(* IEC 61131-3 sources: manufacturing_io/scenes (part 2) *)

(* ---- mps-sorting.st ---- *)
VAR
	START_EDGE : BOOL;
	PB_START_LAST : BOOL;
	STOP_REQ : BOOL;
	SEL_LAST : BOOL := TRUE;
	SEL_CHANGED : BOOL;
	T_WD : TON;
	T_READ : TON;
	T_FEED : TON;
	STEP_LAST : UDINT;
	KIND : UINT;
	NEXT_FEED : UINT;
	CLEAR : BOOL;
	RUNNING : BOOL;
	MEM_BELT : BOOL;
	MEM_STOP : BOOL;
	MEM_W1 : BOOL;
	MEM_W2 : BOOL;
	IND_BELT_LAST : BOOL;
	IND_STOP_LAST : BOOL;
	IND_W1_LAST : BOOL;
	IND_W2_LAST : BOOL;
	IND_ACTIVE : BOOL;
	ESTOP : BOOL;
	READY : BOOL;
	MASTER_ON : BOOL;
	HOMED : BOOL;
	MASTER_EDGE : BOOL;
	PB_MASTER_LAST : BOOL;
	HOME_EDGE : BOOL;
	PB_HOME_LAST : BOOL;
END_VAR
// mps-sorting: Festo Didactic's MPS Sorting station 8046325 (manual 8046391, 11/2015). The
// sequence and the IO are the manual's: a 40 mm workpiece is laid on the belt, a fork light
// barrier sees it, the belt runs it up to a stop, and three sensors at the stop say what it is -
// a through-beam sees every workpiece, a retro-reflective one sees every one that is NOT matt
// black, and an inductive one sees the metal. So black = seen but not by the retro one, red =
// retro but not inductive, metallic = both. Red goes to the chute at the belt START (Weiche 1),
// metallic to the one in the MIDDLE (Weiche 2), black runs off the belt END.
// The same sequence runs without a PLC in mps-sorting.ctl.js - keep the two in step.
//
// ONE difference from the real machine, deliberate: Festo's Q3 is "Stopper einfahren" - the stop
// is out by default and the output retracts it. Here the stop pops UP out of the belt
// (STOP_HOLD, energised to hold), because in this simulator a stop a part passes UNDER holds it
// from a positive distance (CLAUDE.md). It is the same signal inverted.
//
// KIND: 0 = black, 1 = red, 2 = metallic.

START_EDGE := PB_START AND NOT PB_START_LAST;
PB_START_LAST := PB_START;
IF PB_CSTOP THEN
	STOP_REQ := TRUE;
END_IF;
SEL_CHANGED := SEL_AUTO <> SEL_LAST;
SEL_LAST := SEL_AUTO;

ESTOP := PB_ESTOP;
MASTER_EDGE := PB_MASTER AND NOT PB_MASTER_LAST;
PB_MASTER_LAST := PB_MASTER;
HOME_EDGE := PB_HOME AND NOT PB_HOME_LAST;
PB_HOME_LAST := PB_HOME;
IF ESTOP THEN
	MASTER_ON := FALSE;
	HOMED := FALSE;
ELSIF MASTER_EDGE THEN
	MASTER_ON := TRUE;
END_IF;
READY := MASTER_ON AND NOT ESTOP;

// Everything laid on the belt has reached a bin: the invariant a discharge step waits for. A
// count that "has moved" cannot say WHICH workpiece moved (CLAUDE.md).
CLEAR := (EM_BLACK_CNT + EM_RED_CNT + EM_METAL_CNT) = (RM_1_CNT + RM_2_CNT + RM_3_CNT);

CASE ST1_STEP OF
	0:	// Ausgangsstellung: belt off, stop out, both gates in
		BELT_FWD := FALSE;
		W1_EXT := FALSE;
		W2_EXT := FALSE;
		EM_BLACK := FALSE;
		EM_RED := FALSE;
		EM_METAL := FALSE;
		STOP_HOLD := TRUE;
		IF START_EDGE AND SEL_AUTO AND READY AND HOMED THEN
			STOP_REQ := FALSE;
			ST1_STEP := 10;
		END_IF;
	10:	// the operator lays the next workpiece on the belt, one colour at a time
		BELT_FWD := FALSE;
		STOP_HOLD := TRUE;
		EM_BLACK := NEXT_FEED = 0;
		EM_RED := NEXT_FEED = 1;
		EM_METAL := NEXT_FEED = 2;
		IF T_FEED.Q THEN
			NEXT_FEED := (NEXT_FEED + 1) MOD 3;
			ST1_STEP := 15;
		END_IF;
	15:	// Startvoraussetzung: Werkstück am Bandanfang
		EM_BLACK := FALSE;
		EM_RED := FALSE;
		EM_METAL := FALSE;
		BELT_FWD := FALSE;
		STOP_HOLD := TRUE;
		IF WP_AT_START AND NOT CHUTE_FULL THEN
			ST1_STEP := 20;
		END_IF;
	20:	// Bandmotor ein
		BELT_FWD := TRUE;
		STOP_HOLD := TRUE;
		IF WP_DETECTED THEN
			ST1_STEP := 30;
		END_IF;
	30:	// Farb-/Materialidentifikation, with the workpiece held against the stop
		BELT_FWD := TRUE;
		IF T_READ.Q THEN
			IF WP_METALLIC THEN
				KIND := 2;
				ST1_STEP := 50;
			ELSIF WP_NOT_BLACK THEN
				KIND := 1;
				ST1_STEP := 40;
			ELSE
				KIND := 0;
				ST1_STEP := 60;
			END_IF;
		END_IF;
	40:	// red: Weiche 1 ausfahren
		BELT_FWD := TRUE;
		W1_EXT := TRUE;
		IF W1_OUT THEN
			ST1_STEP := 41;
		END_IF;
	41:	// Sperre einfahren
		BELT_FWD := TRUE;
		STOP_HOLD := FALSE;
		IF AS_STOP_FREE THEN
			ST1_STEP := 42;
		END_IF;
	42:	// Werkstück ausgeschleust
		BELT_FWD := TRUE;
		IF CLEAR THEN
			ST1_STEP := 43;
		END_IF;
	43:	// Weiche 1 einfahren
		BELT_FWD := TRUE;
		W1_EXT := FALSE;
		IF AS_W1_IN THEN
			ST1_STEP := 70;
		END_IF;
	50:	// metallic: Weiche 2 ausfahren
		BELT_FWD := TRUE;
		W2_EXT := TRUE;
		IF W2_OUT THEN
			ST1_STEP := 51;
		END_IF;
	51:
		BELT_FWD := TRUE;
		STOP_HOLD := FALSE;
		IF AS_STOP_FREE THEN
			ST1_STEP := 52;
		END_IF;
	52:
		BELT_FWD := TRUE;
		IF CLEAR THEN
			ST1_STEP := 53;
		END_IF;
	53:
		BELT_FWD := TRUE;
		W2_EXT := FALSE;
		IF AS_W2_IN THEN
			ST1_STEP := 70;
		END_IF;
	60:	// black: let it go, it runs off the belt end onto the third chute
		BELT_FWD := TRUE;
		STOP_HOLD := FALSE;
		IF AS_STOP_FREE THEN
			ST1_STEP := 61;
		END_IF;
	61:
		BELT_FWD := TRUE;
		IF CLEAR THEN
			ST1_STEP := 70;
		END_IF;
	70:	// Bandmotor aus, Sperre ausfahren
		BELT_FWD := FALSE;
		STOP_HOLD := TRUE;
		IF AS_STOP_HOLD THEN
			CYCLE_CNT := CYCLE_CNT + 1;
			IF STOP_REQ THEN
				ST1_STEP := 0;
			ELSE
				ST1_STEP := 10;
			END_IF;
		END_IF;
	800:	// HOME is the station's Ausgangsstellung
		BELT_FWD := FALSE;
		W1_EXT := FALSE;
		W2_EXT := FALSE;
		EM_BLACK := FALSE;
		EM_RED := FALSE;
		EM_METAL := FALSE;
		STOP_HOLD := TRUE;
		IF AS_STOP_HOLD AND AS_W1_IN AND AS_W2_IN THEN
			HOMED := TRUE;
			ST1_STEP := 0;
		END_IF;
	900:	// stuck, or the selector was turned while running
		BELT_FWD := FALSE;
		W1_EXT := FALSE;
		W2_EXT := FALSE;
		EM_BLACK := FALSE;
		EM_RED := FALSE;
		EM_METAL := FALSE;
		IF START_EDGE AND SEL_AUTO THEN
			STOP_REQ := FALSE;
			ST1_STEP := 0;
		END_IF;
	910:	// the master circuit is open: the stop KEEPS the workpiece it is holding
		BELT_FWD := FALSE;
		W1_EXT := FALSE;
		W2_EXT := FALSE;
		EM_BLACK := FALSE;
		EM_RED := FALSE;
		EM_METAL := FALSE;
		IF READY THEN
			ST1_STEP := 0;
		END_IF;
END_CASE;

RUNNING := ST1_STEP <> 0 AND ST1_STEP <> 800 AND ST1_STEP <> 900 AND ST1_STEP <> 910;

// TONs after the CASE: their Q is read by the NEXT scan.
T_READ(In := ST1_STEP = 30, PT := T#400ms);
T_FEED(In := ST1_STEP = 10, PT := T#600ms);

// Watchdog: a running step that stops moving is a jam, not patience - a workpiece taken off the
// belt by hand leaves step 20 waiting for a stop it will never reach. The TON is called BEFORE
// STEP_LAST is updated, so a step change gives it one scan of In = FALSE and resets it.
T_WD(In := ST1_STEP <> 0 AND ST1_STEP <> 900 AND ST1_STEP <> 910 AND ST1_STEP = STEP_LAST, PT := T#20s);
STEP_LAST := ST1_STEP;
IF T_WD.Q OR (SEL_CHANGED AND RUNNING) THEN
	ST1_STEP := 900;
	BELT_FWD := FALSE;
	W1_EXT := FALSE;
	W2_EXT := FALSE;
	EM_BLACK := FALSE;
	EM_RED := FALSE;
	EM_METAL := FALSE;
END_IF;

IF ESTOP THEN
	IF ST1_STEP <> 910 THEN
		ST1_STEP := 910;
	END_IF;
	BELT_FWD := FALSE;
	W1_EXT := FALSE;
	W2_EXT := FALSE;
	EM_BLACK := FALSE;
	EM_RED := FALSE;
	EM_METAL := FALSE;
ELSIF HOME_EDGE AND READY AND ST1_STEP = 0 THEN
	ST1_STEP := 800;
END_IF;

AUTO_RUN := ST1_STEP <> 0 AND ST1_STEP <> 800 AND ST1_STEP <> 900 AND ST1_STEP <> 910;
IND_ACTIVE := NOT SEL_AUTO AND NOT AUTO_RUN AND READY AND ST1_STEP <> 800;
IF IND_ACTIVE THEN
	IF IND_BELT AND NOT IND_BELT_LAST THEN
		MEM_BELT := NOT MEM_BELT;
	END_IF;
	IF IND_STOP AND NOT IND_STOP_LAST THEN
		MEM_STOP := NOT MEM_STOP;
	END_IF;
	IF IND_W1 AND NOT IND_W1_LAST THEN
		MEM_W1 := NOT MEM_W1;
	END_IF;
	IF IND_W2 AND NOT IND_W2_LAST THEN
		MEM_W2 := NOT MEM_W2;
	END_IF;
	BELT_FWD := MEM_BELT;
	STOP_HOLD := MEM_STOP;
	W1_EXT := MEM_W1;
	W2_EXT := MEM_W2;
	EM_BLACK := IND_FEED_BLACK;
	EM_RED := IND_FEED_RED;
	EM_METAL := IND_FEED_METAL;
ELSE
	MEM_BELT := FALSE;
	MEM_STOP := FALSE;
	MEM_W1 := FALSE;
	MEM_W2 := FALSE;
END_IF;
IND_BELT_LAST := IND_BELT;
IND_STOP_LAST := IND_STOP;
IND_W1_LAST := IND_W1;
IND_W2_LAST := IND_W2;

OVR := OVR_SET;
PL_START := AUTO_RUN;
PL_MASTER := MASTER_ON;
PL_HOME := HOMED;

(* ---- pallet-line.st ---- *)
VAR
	START_EDGE : BOOL;
	PB_START_LAST : BOOL;
	STOP_REQ : BOOL;
	SEL_LAST : BOOL := TRUE;
	SEL_CHANGED : BOOL;
	T_DWELL : TON;
	T_SETTLE : TON;
	T_CONF : TON;
	T_WD : TON;
	EM_P_LAST : UDINT;
	EM_W_LAST : UDINT;
	STEP_LAST : UDINT;
	GONE : UDINT;
	FED : UDINT;
	MEM_CV : BOOL;
	MEM_STOP : BOOL;
	MEM_LIFT : BOOL;
	IND_CV_LAST : BOOL;
	IND_STOP_LAST : BOOL;
	IND_LIFT_LAST : BOOL;
	ESTOP : BOOL;
	READY : BOOL;
	MASTER_ON : BOOL;
	HOMED : BOOL;
	MASTER_EDGE : BOOL;
	PB_MASTER_LAST : BOOL;
	HOME_EDGE : BOOL;
	PB_HOME_LAST : BOOL;
END_VAR
// pallet-line: a pallet is fed onto the belt, stopped at the station by a POP-UP stop, lifted off
// the belt and located square on its pins, loaded with a part, then put back down and released to
// the unloader. Repeat until CYCLE STOP. The same sequence runs without a PLC in pallet-line.ctl.js.
//
// The stop pops UP from under the belt on purpose. An overhead pin that the pallet has to drive
// under holds it from 7.9-15.1 mm away even after it has lifted clear and come to rest, and the
// clearance sweep is non-monotonic (5.1 held, 8.1 free, 11.1 free, 14.1 HELD, 17.1+ free), so
// there is no clearance to design to. Retracted, a pop-up stop is below the belt surface and
// nothing stands in the path at all.
//
// The pin must also be UP before a pallet arrives: one that rises under a pallet already over it
// tips the pallet off the belt (measured).
//
// The unloader counts the pallet AND the part riding on it, so the discharge step waits on both
// feeders: RM_CNT + GONE >= EM_P_CNT + EM_W_CNT.
//
// The panel has a selector AUTO / INDIVIDUAL (rb4axis): START only in AUTO, the individual buttons
// only in INDIVIDUAL, and a change while the sequence runs is a FAULT, not a pause.

START_EDGE := PB_START AND NOT PB_START_LAST;
PB_START_LAST := PB_START;
IF PB_CSTOP THEN
	STOP_REQ := TRUE;
END_IF;
SEL_CHANGED := SEL_AUTO <> SEL_LAST;
SEL_LAST := SEL_AUTO;

// The master circuit, as on the cell panel: E-STOP is a latching mushroom, MASTER ON energises
// the machine, and nothing runs without it. An E-STOP also loses the home position.
ESTOP := PB_ESTOP;
MASTER_EDGE := PB_MASTER AND NOT PB_MASTER_LAST;
PB_MASTER_LAST := PB_MASTER;
HOME_EDGE := PB_HOME AND NOT PB_HOME_LAST;
PB_HOME_LAST := PB_HOME;
IF ESTOP THEN
	MASTER_ON := FALSE;
	HOMED := FALSE;
ELSIF MASTER_EDGE THEN
	MASTER_ON := TRUE;
END_IF;
READY := MASTER_ON AND NOT ESTOP;

FED := EM_P_CNT + EM_W_CNT;
// A write-off goes STALE when what was written off turns up after all. GONE is a UDINT, so
// FED - RM_CNT with RM ahead underflows to about 4 billion: guard before you subtract.
IF RM_CNT >= FED THEN
	GONE := 0;
ELSIF RM_CNT + GONE > FED THEN
	GONE := FED - RM_CNT;
END_IF;

CASE ST1_STEP OF
	0:	// idle
		CV1_RUN := FALSE;
		EM_P_EMIT := FALSE;
		EM_W_EMIT := FALSE;
		SOL_LIFT := FALSE;
		SOL_STOP := FALSE;
		IF START_EDGE AND SEL_AUTO AND READY AND HOMED AND AS_LIFT_DN THEN
			STOP_REQ := FALSE;
			ST1_STEP := 10;
		END_IF;
	10:	// stop UP first, before any pallet is on its way
		SOL_STOP := TRUE;
		IF AS_STOP_UP THEN
			EM_P_LAST := EM_P_CNT;
			ST1_STEP := 20;
		END_IF;
	20:	// feed one pallet
		CV1_RUN := TRUE;
		EM_P_EMIT := TRUE;
		IF EM_P_CNT <> EM_P_LAST THEN
			EM_P_EMIT := FALSE;
			ST1_STEP := 30;
		END_IF;
	30:	// convey it to the station. The beam only says a pallet is HERE; the PIN locates it.
		// Stopping the belt on the beam edge left the pallet 106 mm short of the pin, so the
		// part feeder dropped its load onto the belt behind the deck every cycle (measured).
		CV1_RUN := TRUE;
		IF PE_STN THEN
			ST1_STEP := 35;
		END_IF;
	35:	// keep driving until it is pressed against the pin
		CV1_RUN := TRUE;
		IF T_SETTLE.Q THEN
			CV1_RUN := FALSE;
			ST1_STEP := 40;
		END_IF;
	40:	// lift and locate. The pallet must stay reported present for a CONFIRM time, not just for
		// the instant the switch first makes: a part is dropped on the strength of this signal,
		// and T_CONF restarts if it flickers.
		SOL_LIFT := TRUE;
		IF T_CONF.Q THEN
			EM_W_LAST := EM_W_CNT;
			ST1_STEP := 50;
		END_IF;
	50:	// load one part onto the pallet
		EM_W_EMIT := TRUE;
		IF EM_W_CNT <> EM_W_LAST THEN
			EM_W_EMIT := FALSE;
			ST1_STEP := 60;
		END_IF;
	60:	// the station does its work
		IF T_DWELL.Q THEN
			ST1_STEP := 70;
		END_IF;
	70:	// pallet back onto the belt
		SOL_LIFT := FALSE;
		IF AS_LIFT_DN THEN
			ST1_STEP := 80;
		END_IF;
	80:	// only now is the pin allowed down, clear of the path
		SOL_STOP := FALSE;
		IF AS_STOP_DN THEN
			ST1_STEP := 90;
		END_IF;
	90:	// discharge: every pallet and part fed must have reached the unloader
		CV1_RUN := TRUE;
		IF RM_CNT + GONE >= FED THEN
			CV1_RUN := FALSE;
			ST1_STEP := 100;
		END_IF;
	100:	// cycle complete
		CYCLE_CNT := CYCLE_CNT + 1;
		IF STOP_REQ THEN
			ST1_STEP := 0;
		ELSE
			ST1_STEP := 10;
		END_IF;
	800:	// HOME: the lift down and the pin down, so the belt is clear along its whole length
		CV1_RUN := FALSE;
		EM_P_EMIT := FALSE;
		EM_W_EMIT := FALSE;
		SOL_LIFT := FALSE;
		SOL_STOP := FALSE;
		IF AS_LIFT_DN AND AS_STOP_DN THEN
			HOMED := TRUE;
			ST1_STEP := 0;
		END_IF;
	910:	// E-STOP: the master circuit is open, so every solenoid de-energises - a 5/2 single-
		// solenoid valve springs back. The LIFT is the exception: it is a holder, and a real
		// machine does not drop what it carries when the power goes.
		CV1_RUN := FALSE;
		EM_P_EMIT := FALSE;
		EM_W_EMIT := FALSE;
		SOL_STOP := FALSE;
		IF READY THEN	// MASTER ON after the mushroom is released
			ST1_STEP := 0;
		END_IF;
	900:	// FAULT: a step stopped moving. Stop feeding and the belt; the pin keeps holding the
		// queue back and the lift keeps its pallet.
		CV1_RUN := FALSE;
		EM_P_EMIT := FALSE;
		EM_W_EMIT := FALSE;
		IF START_EDGE AND SEL_AUTO THEN
			STOP_REQ := FALSE;
			// Acknowledging writes off what never reached the unloader. Only HERE: at every START
			// it would write off pallets still legitimately on the belt.
			GONE := FED - RM_CNT;
			ST1_STEP := 0;
		END_IF;
END_CASE;

T_DWELL(In := (ST1_STEP = 60), PT := T#500ms);
// 106 mm from the beam edge to the pin at 250 mm/s is 424 ms; 700 leaves margin to press up.
T_SETTLE(In := (ST1_STEP = 35), PT := T#700ms);
T_CONF(In := (ST1_STEP = 40) AND AS_LIFT_UP AND PLT_PRESENT, PT := T#300ms);

// Watchdog: a running step that stops moving is a jam, not patience. Without it the sequence waits
// for ever and the machine only LOOKS alive. A selector change while running trips the same way.
T_WD(In := (ST1_STEP = STEP_LAST) AND (ST1_STEP <> 0) AND (ST1_STEP <> 900) AND (ST1_STEP <> 910), PT := T#15s);
IF ST1_STEP <> STEP_LAST THEN
	STEP_LAST := ST1_STEP;
END_IF;
IF T_WD.Q OR (SEL_CHANGED AND (ST1_STEP <> 0) AND (ST1_STEP <> 900) AND (ST1_STEP <> 910)) THEN
	ST1_STEP := 900;
	CV1_RUN := FALSE;
	EM_P_EMIT := FALSE;
	EM_W_EMIT := FALSE;
END_IF;

// E-STOP at any moment, and the HOME button when the machine is energised and idle.
IF ESTOP THEN
	IF ST1_STEP <> 910 THEN
		ST1_STEP := 910;
	END_IF;
	CV1_RUN := FALSE;
	EM_P_EMIT := FALSE;
	EM_W_EMIT := FALSE;
	SOL_STOP := FALSE;
ELSIF HOME_EDGE AND READY AND (ST1_STEP = 0) THEN
	ST1_STEP := 800;
END_IF;

AUTO_RUN := (ST1_STEP <> 0) AND (ST1_STEP <> 800) AND (ST1_STEP <> 900) AND (ST1_STEP <> 910);

// Individual operation: the buttons are momentary; the PLC keeps a toggle memory per actuator and
// clears it when INDIVIDUAL ends, so nothing stays latched into AUTO.
IF NOT SEL_AUTO AND NOT AUTO_RUN AND READY AND (ST1_STEP <> 800) THEN
	IF IND_CV AND NOT IND_CV_LAST THEN
		MEM_CV := NOT MEM_CV;
	END_IF;
	IF IND_STOP AND NOT IND_STOP_LAST THEN
		MEM_STOP := NOT MEM_STOP;
	END_IF;
	IF IND_LIFT AND NOT IND_LIFT_LAST THEN
		MEM_LIFT := NOT MEM_LIFT;
	END_IF;
	CV1_RUN := MEM_CV;
	SOL_STOP := MEM_STOP;
	SOL_LIFT := MEM_LIFT;
	EM_P_EMIT := IND_FEED_P;
	EM_W_EMIT := IND_FEED_W;
ELSE
	MEM_CV := FALSE;
	MEM_STOP := FALSE;
	MEM_LIFT := FALSE;
END_IF;
IND_CV_LAST := IND_CV;
IND_STOP_LAST := IND_STOP;
IND_LIFT_LAST := IND_LIFT;

// The speed override the operator dialled in, passed on to the axes and the belts.
OVR := OVR_SET;

PL_START := AUTO_RUN;
PL_MASTER := MASTER_ON;
PL_HOME := HOMED;

(* ---- palletizing.st ---- *)
VAR
	START_EDGE : BOOL;
	PB_START_LAST : BOOL;
	STOP_REQ : BOOL;
	SEL_LAST : BOOL := TRUE;
	SEL_CHANGED : BOOL;
	ESTOP : BOOL;
	READY : BOOL;
	MASTER_ON : BOOL;
	HOMED : BOOL;
	MASTER_EDGE : BOOL;
	PB_MASTER_LAST : BOOL;
	HOME_EDGE : BOOL;
	PB_HOME_LAST : BOOL;
	RUNNING : BOOL;
	LOAD_BUSY : BOOL;
	UNLOAD_BUSY : BOOL;
	LOAD_IDX : INT;
	UNLOAD_IDX : INT;
	FULL : ARRAY[0..3] OF BOOL;
	HALF : BOOL;
	ROW_Y : LREAL := 330.0;
	PICKED : BOOL;
	ANY_VAC : BOOL;
	NO_VAC : BOOL;
	NO_UVAC : BOOL;
	NEED_FILL : BOOL := TRUE;
	PAL_BASE : UDINT;
	NEXT_ST : INT;
	T_FILL : TON;
	T_PICK : TON;
	T_UPICK : TON;
	T_WD1 : TON;
	T_WD2 : TON;
	T_WD3 : TON;
	STEP1_LAST : UDINT;
	STEP2_LAST : UDINT;
	STEP3_LAST : UDINT;
	JAM : BOOL;
	MEM_VAC : BOOL;
	IND_VAC_LAST : BOOL;
	MEM_LIFT : BOOL;
	IND_LIFT_LAST : BOOL;
	MEM_PAL : BOOL;
	IND_PAL_LAST : BOOL;
	MEM_JIG : BOOL;
	IND_JIG_LAST : BOOL;
	MEM_UVAC : BOOL;
	IND_UVAC_LAST : BOOL;
	MEM_ULIFT : BOOL;
	IND_ULIFT_LAST : BOOL;
	MEM_USHIFT : BOOL;
	IND_USHIFT_LAST : BOOL;
	INDIVIDUAL : BOOL;
END_VAR
// palletizing: a 10 x 10 pallet of spark plugs, a five-up vacuum gantry on two servo axes, a
// rotary carrier of five-slot jigs, and an unload head that hands the plugs to the next process.
// The same sequence runs without a PLC in palletizing.ctl.js.
//
// THREE stations run at the same time, which is what a cell does and what one long sequence could
// not: the gantry goes back for the next five as soon as it has put its five down, while the
// carrier indexes and the unloader empties a jig on the far side. They meet at the carrier: FULL[i]
// says which jig has parts in it, and neither head lets the table turn under it.
//
// A head takes what is there. A hole may be empty - a plug was lifted out, or the pallet is
// finished - and the gantry carries on with what it got rather than waiting for a plug that is not
// coming. Nothing at all means the tray is empty, and a fresh pallet is called for.
//
// Gantry positions are millimetres on each axis, measured from the scene: cup 3 sits at
// X = GX - 300 and Y = GY - 600, so the pallet halves are at GX 150 and 450, the jig at GX 1268,
// and pallet row r is at GY 330 + 60 r.

START_EDGE := PB_START AND NOT PB_START_LAST;
PB_START_LAST := PB_START;
IF PB_CSTOP THEN
	STOP_REQ := TRUE;
END_IF;
SEL_CHANGED := SEL_AUTO <> SEL_LAST;
SEL_LAST := SEL_AUTO;

// The master circuit: E-STOP is a latching mushroom, MASTER ON energises the machine, and an
// E-STOP also loses the home position.
ESTOP := PB_ESTOP;
MASTER_EDGE := PB_MASTER AND NOT PB_MASTER_LAST;
PB_MASTER_LAST := PB_MASTER;
HOME_EDGE := PB_HOME AND NOT PB_HOME_LAST;
PB_HOME_LAST := PB_HOME;
IF ESTOP THEN
	MASTER_ON := FALSE;
	HOMED := FALSE;
ELSIF MASTER_EDGE THEN
	MASTER_ON := TRUE;
END_IF;
READY := MASTER_ON AND NOT ESTOP;

ANY_VAC := VAC_SW1 OR VAC_SW2 OR VAC_SW3 OR VAC_SW4 OR VAC_SW5;
NO_VAC := NOT ANY_VAC;
NO_UVAC := NOT (UVAC_SW1 OR UVAC_SW2 OR UVAC_SW3 OR UVAC_SW4 OR UVAC_SW5);
// The jig standing at the load station, and the one at the unload station.
LOAD_IDX := (2 - TBL_STATION + 4) MOD 4;
UNLOAD_IDX := (4 - TBL_STATION) MOD 4;
// Neither head lets the carrier turn while it is over a jig.
LOAD_BUSY := (ST1_STEP >= 57) AND (ST1_STEP <= 80);
UNLOAD_BUSY := (ST3_STEP >= 110) AND (ST3_STEP <= 130);

// ---------------------------------------------------------------- ST1: the depalletiser
CASE ST1_STEP OF
	0:	// idle: head up, vacuum off
		VAC_ON := FALSE;
		GX_EXEC := FALSE;
		GY_EXEC := FALSE;
		SOL_Z_DN := FALSE;
		SOL_Z_UP := TRUE;
		EM_PAL_EN := FALSE;
		IF START_EDGE AND SEL_AUTO AND READY AND HOMED AND AS_Z_UP AND AS_U_UP THEN
			STOP_REQ := FALSE;
			ST2_STEP := 10;
			ST3_STEP := 100;
			IF NEED_FILL THEN
				PAL_BASE := EM_PAL_CNT;
				ST1_STEP := 5;
			ELSE
				ST1_STEP := 10;
			END_IF;
		END_IF;
	5:	// A fresh pallet. The tray is FULL when the loader stops delivering, not after a count of
		// 100: a hole that still had a plug in it would make a count wait for ever.
		PAL_CLAMP := TRUE;
		EM_PAL_EN := TRUE;
		IF EM_PAL_CNT <> PAL_BASE THEN
			PAL_BASE := EM_PAL_CNT;
		ELSIF T_FILL.Q THEN
			EM_PAL_EN := FALSE;
			NEED_FILL := FALSE;
			ST1_STEP := 10;
		END_IF;
	10:	// both gantry axes move at once; Execute is a LEVEL held until Done
		PAL_CLAMP := TRUE;
		JIG_CLAMP := TRUE;
		IF HALF THEN
			GX_TGT := 450.0;
		ELSE
			GX_TGT := 150.0;
		END_IF;
		GY_TGT := ROW_Y;
		GX_EXEC := TRUE;
		GY_EXEC := TRUE;
		IF GX_DONE AND GY_DONE THEN
			GX_EXEC := FALSE;
			GY_EXEC := FALSE;
			ST1_STEP := 15;
		END_IF;
	15:	// wait until the plant has seen Execute drop
		IF NOT GX_DONE AND NOT GY_DONE THEN
			ST1_STEP := 20;
		END_IF;
	20:	// head down onto the row
		SOL_Z_UP := FALSE;
		SOL_Z_DN := TRUE;
		IF AS_Z_DN THEN
			ST1_STEP := 30;
		END_IF;
	30:	// the tray lets go while the cups take whatever is there
		PAL_CLAMP := FALSE;
		VAC_ON := TRUE;
		IF T_PICK.Q THEN
			PICKED := ANY_VAC;
			ST1_STEP := 40;
		END_IF;
	40:	// the tray is held again, and the head lifts with what it got
		PAL_CLAMP := TRUE;
		SOL_Z_DN := FALSE;
		SOL_Z_UP := TRUE;
		IF AS_Z_UP THEN
			IF PICKED THEN
				ST1_STEP := 50;
			ELSE
				// nothing at all came up: the tray is empty
				NEED_FILL := TRUE;
				PAL_BASE := EM_PAL_CNT;
				ST1_STEP := 5;
			END_IF;
		END_IF;
	50:	// across to the jig at the load station
		GX_TGT := 1268.0;
		GY_TGT := 600.0;
		GX_EXEC := TRUE;
		GY_EXEC := TRUE;
		IF GX_DONE AND GY_DONE THEN
			GX_EXEC := FALSE;
			GY_EXEC := FALSE;
			ST1_STEP := 55;
		END_IF;
	55:	// wait until the plant has seen Execute drop
		IF NOT GX_DONE AND NOT GY_DONE THEN
			ST1_STEP := 57;
		END_IF;
	57:	// the load station must be standing still with an empty jig under it
		IF TBL_INPOS AND NOT FULL[LOAD_IDX] THEN
			ST1_STEP := 60;
		END_IF;
	60:	// head down over the jig
		SOL_Z_UP := FALSE;
		SOL_Z_DN := TRUE;
		IF AS_Z_DN THEN
			ST1_STEP := 70;
		END_IF;
	70:	// the jig nests take the plugs as the cups let go: one part, one holder
		VAC_ON := FALSE;
		IF NO_VAC THEN
			ST1_STEP := 80;
		END_IF;
	80:	// head up; the carrier may take this jig away now
		SOL_Z_DN := FALSE;
		SOL_Z_UP := TRUE;
		IF AS_Z_UP THEN
			FULL[LOAD_IDX] := TRUE;
			CYCLE_CNT := CYCLE_CNT + 1;
			IF HALF THEN
				HALF := FALSE;
				IF ROW_Y >= 870.0 THEN
					ROW_Y := 330.0;
					NEED_FILL := TRUE;
				ELSE
					ROW_Y := ROW_Y + 60.0;
				END_IF;
			ELSE
				HALF := TRUE;
			END_IF;
			IF STOP_REQ THEN
				ST1_STEP := 0;
			ELSIF NEED_FILL THEN
				PAL_BASE := EM_PAL_CNT;
				ST1_STEP := 5;
			ELSE
				ST1_STEP := 10;
			END_IF;
		END_IF;
	800:	// HOME: heads up, unload shift over the jig, both gantry axes to zero, carrier to its
		// origin. The vacuum is left alone: a head keeps the plugs it is holding.
		TBL_RUN := NOT TBL_ORIGIN;
		SOL_Z_DN := FALSE;
		SOL_Z_UP := TRUE;
		SOL_U_DN := FALSE;
		SOL_U_UP := TRUE;
		SOL_U_BIN := FALSE;
		SOL_U_JIG := TRUE;
		GX_TGT := 0.0;
		GY_TGT := 0.0;
		GX_EXEC := TRUE;
		GY_EXEC := TRUE;
		IF AS_Z_UP AND AS_U_UP AND AS_U_JIG AND GX_DONE AND GY_DONE AND TBL_ORIGIN THEN
			GX_EXEC := FALSE;
			GY_EXEC := FALSE;
			TBL_RUN := FALSE;
			HOMED := TRUE;
			ST1_STEP := 0;
		END_IF;
	900:	// FAULT: stuck, or the selector was turned while running. Motion and feeding off; the
		// trays and the cups keep whatever they hold.
		TBL_RUN := FALSE;
		GX_EXEC := FALSE;
		GY_EXEC := FALSE;
		EM_PAL_EN := FALSE;
		PAL_CLAMP := TRUE;
		JIG_CLAMP := TRUE;
		IF START_EDGE AND SEL_AUTO THEN
			STOP_REQ := FALSE;
			ST1_STEP := 0;
		END_IF;
	910:	// E-STOP: the master circuit is open, so every solenoid de-energises - which is what
		// really happens: a 5/2 single-solenoid valve springs back, a double one holds. The trays
		// and the cups KEEP their parts: a hundred plugs let loose in their pockets is not what a
		// power cut does, and it costs the plant four times the work.
		TBL_RUN := FALSE;
		GX_EXEC := FALSE;
		GY_EXEC := FALSE;
		EM_PAL_EN := FALSE;
		SOL_Z_DN := FALSE;
		SOL_Z_UP := FALSE;
		SOL_U_DN := FALSE;
		SOL_U_UP := FALSE;
		SOL_U_BIN := FALSE;
		SOL_U_JIG := FALSE;
		PAL_CLAMP := TRUE;
		JIG_CLAMP := TRUE;
		IF READY THEN	// MASTER ON after the mushroom is released
			ST1_STEP := 0;
		END_IF;
END_CASE;

RUNNING := (ST1_STEP <> 0) AND (ST1_STEP <> 800) AND (ST1_STEP <> 900) AND (ST1_STEP <> 910);

// ---------------------------------------------------------------- ST2: the jig carrier
IF NOT RUNNING THEN
	ST2_STEP := 0;
	TBL_RUN := FALSE;
ELSE
	CASE ST2_STEP OF
		10:	// Turn when there is a full jig to move on AND an empty one to bring to the unloader,
			// and never while a head is over the table.
			TBL_RUN := FALSE;
			IF FULL[LOAD_IDX] AND NOT FULL[UNLOAD_IDX] AND NOT LOAD_BUSY AND NOT UNLOAD_BUSY AND TBL_INPOS THEN
				NEXT_ST := (TBL_STATION + 1) MOD 4;
				ST2_STEP := 20;
			END_IF;
		20:	// the invariant: this index has landed on the station it was sent to
			TBL_RUN := TRUE;
			IF TBL_INPOS AND (TBL_STATION = NEXT_ST) THEN
				TBL_RUN := FALSE;
				ST2_STEP := 10;
			END_IF;
		ELSE
			ST2_STEP := 10;
	END_CASE;
END_IF;

// ---------------------------------------------------------------- ST3: the unloader
IF NOT RUNNING THEN
	ST3_STEP := 0;
ELSE
	CASE ST3_STEP OF
		100:	// wait for a full jig to arrive and stand still
			IF FULL[UNLOAD_IDX] AND TBL_INPOS THEN
				ST3_STEP := 110;
			END_IF;
		110:	// over the jig
			SOL_U_BIN := FALSE;
			SOL_U_JIG := TRUE;
			IF AS_U_JIG THEN
				ST3_STEP := 115;
			END_IF;
		115:	// down onto it
			SOL_U_UP := FALSE;
			SOL_U_DN := TRUE;
			IF AS_U_DN THEN
				ST3_STEP := 120;
			END_IF;
		120:	// whatever is in the jig, however many: a gap is not a reason to stop
			JIG_CLAMP := FALSE;
			UVAC_ON := TRUE;
			IF T_UPICK.Q THEN
				ST3_STEP := 130;
			END_IF;
		130:	// up, and the carrier is free to turn again
			JIG_CLAMP := TRUE;
			SOL_U_DN := FALSE;
			SOL_U_UP := TRUE;
			IF AS_U_UP THEN
				FULL[UNLOAD_IDX] := FALSE;
				ST3_STEP := 140;
			END_IF;
		140:	// across to the next process
			SOL_U_JIG := FALSE;
			SOL_U_BIN := TRUE;
			IF AS_U_BIN THEN
				ST3_STEP := 150;
			END_IF;
		150:	// down over the bin
			SOL_U_UP := FALSE;
			SOL_U_DN := TRUE;
			IF AS_U_DN THEN
				ST3_STEP := 160;
			END_IF;
		160:	// let them go: the next process takes them from here
			UVAC_ON := FALSE;
			IF NO_UVAC THEN
				ST3_STEP := 170;
			END_IF;
		170:	// up
			SOL_U_DN := FALSE;
			SOL_U_UP := TRUE;
			IF AS_U_UP THEN
				ST3_STEP := 180;
			END_IF;
		180:	// back over the jig, ready for the next one
			SOL_U_BIN := FALSE;
			SOL_U_JIG := TRUE;
			IF AS_U_JIG THEN
				ST3_STEP := 100;
			END_IF;
		ELSE
			ST3_STEP := 100;
	END_CASE;
END_IF;

// The loader drops one every 40 ms while it can, so 600 ms of nothing means the tray is full.
T_FILL(In := (ST1_STEP = 5) AND (EM_PAL_CNT = PAL_BASE), PT := T#600ms);
// A head is given this long to get hold of what is under it, then carries on with what it has.
T_PICK(In := (ST1_STEP = 30), PT := T#600ms);
T_UPICK(In := (ST3_STEP = 120), PT := T#600ms);

// Watchdog, one per station: a running step that stops moving is a jam, not patience. The
// carrier's wait for work and the unloader's wait for a jig are not stuck, so they are excluded.
T_WD1(In := (ST1_STEP = STEP1_LAST) AND RUNNING, PT := T#15s);
T_WD2(In := (ST2_STEP = STEP2_LAST) AND RUNNING AND (ST2_STEP <> 10), PT := T#15s);
T_WD3(In := (ST3_STEP = STEP3_LAST) AND RUNNING AND (ST3_STEP <> 100), PT := T#15s);
IF ST1_STEP <> STEP1_LAST THEN
	STEP1_LAST := ST1_STEP;
END_IF;
IF ST2_STEP <> STEP2_LAST THEN
	STEP2_LAST := ST2_STEP;
END_IF;
IF ST3_STEP <> STEP3_LAST THEN
	STEP3_LAST := ST3_STEP;
END_IF;
JAM := T_WD1.Q OR T_WD2.Q OR T_WD3.Q;
IF RUNNING AND (JAM OR SEL_CHANGED) THEN
	ST1_STEP := 900;
	ST2_STEP := 0;
	ST3_STEP := 0;
	TBL_RUN := FALSE;
	GX_EXEC := FALSE;
	GY_EXEC := FALSE;
	EM_PAL_EN := FALSE;
END_IF;

// E-STOP at any moment, and the HOME button when the machine is energised and idle.
IF ESTOP THEN
	IF ST1_STEP <> 910 THEN
		ST1_STEP := 910;
	END_IF;
	ST2_STEP := 0;
	ST3_STEP := 0;
	TBL_RUN := FALSE;
	GX_EXEC := FALSE;
	GY_EXEC := FALSE;
	EM_PAL_EN := FALSE;
	SOL_Z_DN := FALSE;
	SOL_Z_UP := FALSE;
	SOL_U_DN := FALSE;
	SOL_U_UP := FALSE;
	SOL_U_BIN := FALSE;
	SOL_U_JIG := FALSE;
	PAL_CLAMP := TRUE;
	JIG_CLAMP := TRUE;
ELSIF HOME_EDGE AND READY AND (ST1_STEP = 0) THEN
	ST1_STEP := 800;
END_IF;

AUTO_RUN := (ST1_STEP <> 0) AND (ST1_STEP <> 800) AND (ST1_STEP <> 900) AND (ST1_STEP <> 910);

// Individual operation: momentary buttons, a PLC toggle memory per actuator, cleared when
// INDIVIDUAL ends. The index button is held and the carrier turns while it is down.
INDIVIDUAL := NOT SEL_AUTO AND NOT AUTO_RUN AND READY AND (ST1_STEP <> 800);
IF INDIVIDUAL THEN
	IF IND_VAC AND NOT IND_VAC_LAST THEN
		MEM_VAC := NOT MEM_VAC;
	END_IF;
	IF IND_LIFT AND NOT IND_LIFT_LAST THEN
		MEM_LIFT := NOT MEM_LIFT;
	END_IF;
	IF IND_PAL AND NOT IND_PAL_LAST THEN
		MEM_PAL := NOT MEM_PAL;
	END_IF;
	IF IND_JIG AND NOT IND_JIG_LAST THEN
		MEM_JIG := NOT MEM_JIG;
	END_IF;
	IF IND_UVAC AND NOT IND_UVAC_LAST THEN
		MEM_UVAC := NOT MEM_UVAC;
	END_IF;
	IF IND_ULIFT AND NOT IND_ULIFT_LAST THEN
		MEM_ULIFT := NOT MEM_ULIFT;
	END_IF;
	IF IND_USHIFT AND NOT IND_USHIFT_LAST THEN
		MEM_USHIFT := NOT MEM_USHIFT;
	END_IF;
	VAC_ON := MEM_VAC;
	UVAC_ON := MEM_UVAC;
	PAL_CLAMP := MEM_PAL;
	JIG_CLAMP := MEM_JIG;
	SOL_Z_DN := MEM_LIFT;
	SOL_Z_UP := NOT MEM_LIFT;
	SOL_U_DN := MEM_ULIFT;
	SOL_U_UP := NOT MEM_ULIFT;
	SOL_U_BIN := MEM_USHIFT;
	SOL_U_JIG := NOT MEM_USHIFT;
	TBL_RUN := IND_INDEX;
ELSE
	MEM_VAC := FALSE;
	MEM_LIFT := FALSE;
	MEM_PAL := FALSE;
	MEM_JIG := FALSE;
	MEM_UVAC := FALSE;
	MEM_ULIFT := FALSE;
	MEM_USHIFT := FALSE;
END_IF;
IND_VAC_LAST := IND_VAC;
IND_LIFT_LAST := IND_LIFT;
IND_PAL_LAST := IND_PAL;
IND_JIG_LAST := IND_JIG;
IND_UVAC_LAST := IND_UVAC;
IND_ULIFT_LAST := IND_ULIFT;
IND_USHIFT_LAST := IND_USHIFT;

// The speed override the operator dialled in, passed on to the axes and the belts.
OVR := OVR_SET;

// Jog: the axis creeps while the button is held, and only on INDIVIDUAL.
GX_JOG_P := INDIVIDUAL AND IND_GX_P;
GX_JOG_N := INDIVIDUAL AND IND_GX_N;
GY_JOG_P := INDIVIDUAL AND IND_GY_P;
GY_JOG_N := INDIVIDUAL AND IND_GY_N;

PL_START := AUTO_RUN;
PL_MASTER := MASTER_ON;
PL_HOME := HOMED;

(* ---- pick-place.st ---- *)
VAR
	START_EDGE : BOOL;
	PB_START_LAST : BOOL;
	STOP_REQ : BOOL;
	T_WD : TON;
	EM_LAST : UDINT;
	STEP_LAST : UDINT;
	GONE : UDINT;
END_VAR
// pick-place: feed a part into the pick nest, pick it with the vacuum cup on the lift cylinder,
// traverse on the servo, lay it on the running outfeed belt, and come home while the belt takes
// it to the unloader. Repeat until STOP. The same sequence runs without a PLC in
// pick-place.ctl.js.
//
// Two handshakes matter. The servo's Execute is a LEVEL held until Done, and Done must be seen
// to drop before the next Execute. The nest clamp must open BEFORE the cup can take the part:
// one part is held by one holder.
//
// Waiting steps wait for an INVARIANT, not for a counter to move: a change cannot say which
// part moved (measured on a-to-b against the simulator: parts piled up, then pipelined).

START_EDGE := PB_START AND NOT PB_START_LAST;
PB_START_LAST := PB_START;
IF PB_STOP THEN
	STOP_REQ := TRUE;
END_IF;

// A write-off goes STALE when the part turns up after all, and then RM + GONE runs PAST EM and
// step 130 stops waiting at all. GONE is a UDINT, so EM_CNT - RM_CNT with RM ahead underflows to
// about 4 billion: guard before you subtract.
IF RM_CNT >= EM_CNT THEN
	GONE := 0;
ELSIF RM_CNT + GONE > EM_CNT THEN
	GONE := EM_CNT - RM_CNT;
END_IF;

CASE ST1_STEP OF
	0:	// idle
		CV_RUN := FALSE;
		EM_EMIT := FALSE;
		VAC_ON := FALSE;
		SOL_Z_DN := FALSE;
		SOL_Z_UP := TRUE;
		SV_EXEC := FALSE;
		IF START_EDGE AND AS_Z_UP AND SV_INPOS AND NOT SV_DONE THEN
			STOP_REQ := FALSE;
			EM_LAST := EM_CNT;
			ST1_STEP := 10;
		END_IF;
	10:	// belt on, feed one part
		CV_RUN := TRUE;
		CLAMP_A := TRUE;
		EM_EMIT := TRUE;
		IF EM_CNT <> EM_LAST THEN
			EM_EMIT := FALSE;
			ST1_STEP := 20;
		END_IF;
	20:	// the nest reports the part
		IF NEST_A_P THEN
			ST1_STEP := 30;
		END_IF;
	30:	// lift down onto the part
		SOL_Z_UP := FALSE;
		SOL_Z_DN := TRUE;
		IF AS_Z_DN THEN
			ST1_STEP := 40;
		END_IF;
	40:	// nest lets go, vacuum takes over
		CLAMP_A := FALSE;
		VAC_ON := TRUE;
		IF VAC_SW THEN
			ST1_STEP := 50;
		END_IF;
	50:	// lift up with the part
		SOL_Z_DN := FALSE;
		SOL_Z_UP := TRUE;
		IF AS_Z_UP THEN
			ST1_STEP := 60;
		END_IF;
	60:	// traverse to the belt
		SV_TGT := 600.0;
		SV_EXEC := TRUE;
		IF SV_DONE THEN
			SV_EXEC := FALSE;
			ST1_STEP := 70;
		END_IF;
	70:	// wait until the plant has seen Execute drop
		IF NOT SV_DONE THEN
			ST1_STEP := 80;
		END_IF;
	80:	// lift down over the belt
		SOL_Z_UP := FALSE;
		SOL_Z_DN := TRUE;
		IF AS_Z_DN THEN
			ST1_STEP := 90;
		END_IF;
	90:	// let the part go onto the belt
		VAC_ON := FALSE;
		IF NOT VAC_SW THEN
			ST1_STEP := 100;
		END_IF;
	100:	// lift up
		SOL_Z_DN := FALSE;
		SOL_Z_UP := TRUE;
		IF AS_Z_UP THEN
			ST1_STEP := 110;
		END_IF;
	110:	// traverse home
		SV_TGT := 0.0;
		SV_EXEC := TRUE;
		IF SV_DONE THEN
			SV_EXEC := FALSE;
			ST1_STEP := 120;
		END_IF;
	120:	// wait until the plant has seen Execute drop
		IF NOT SV_DONE THEN
			ST1_STEP := 130;
		END_IF;
	130:	// the belt carries the part to the unloader: everything loaded must have left
		IF RM_CNT + GONE >= EM_CNT THEN
			CYCLE_CNT := CYCLE_CNT + 1;
			IF STOP_REQ THEN
				ST1_STEP := 0;
			ELSE
				EM_LAST := EM_CNT;
				ST1_STEP := 10;
			END_IF;
		END_IF;
	900:	// FAULT: a step stopped moving. Stop feeding and the servo, but KEEP vacuum: a real
		// machine does not drop the part it is holding.
		EM_EMIT := FALSE;
		CV_RUN := FALSE;
		SV_EXEC := FALSE;
		IF START_EDGE THEN
			STOP_REQ := FALSE;
			// Acknowledging writes off whatever never reached the unloader. Only HERE: at every
			// START it would write off parts still legitimately in the machine, and then an older
			// part's removal ends this cycle - the pipelining bug that cost two live rounds.
			GONE := EM_CNT - RM_CNT;
			ST1_STEP := 0;
		END_IF;
END_CASE;

// Watchdog: a step that stops moving is a jam, not patience. Measured before this existed: taking
// the part out of the nest left ST1_STEP at 20 indefinitely with AUTO_RUN still on.
T_WD(In := (ST1_STEP = STEP_LAST) AND (ST1_STEP <> 0) AND (ST1_STEP <> 900), PT := T#15s);
IF ST1_STEP <> STEP_LAST THEN
	STEP_LAST := ST1_STEP;
END_IF;
IF T_WD.Q THEN
	ST1_STEP := 900;
	EM_EMIT := FALSE;
	CV_RUN := FALSE;
	SV_EXEC := FALSE;
END_IF;

AUTO_RUN := (ST1_STEP <> 0) AND (ST1_STEP <> 900);
PL_START := AUTO_RUN;

(* ---- press-station.st ---- *)
VAR
	START_EDGE : BOOL;
	PB_START_LAST : BOOL;
	STOP_REQ : BOOL;
	SEL_LAST : BOOL := TRUE;
	SEL_CHANGED : BOOL;
	EM_LAST : UDINT;
	T_PRESS : TON;
	T_WD : TON;
	STEP_LAST : UDINT;
	GONE : UDINT;
	MEM_CLAMP : BOOL;
	IND_CLAMP_LAST : BOOL;
	MEM_PRESS : BOOL;
	IND_PRESS_LAST : BOOL;
	MEM_EJECT : BOOL;
	IND_EJECT_LAST : BOOL;
	ESTOP : BOOL;
	READY : BOOL;
	MASTER_ON : BOOL;
	HOMED : BOOL;
	MASTER_EDGE : BOOL;
	PB_MASTER_LAST : BOOL;
	HOME_EDGE : BOOL;
	PB_HOME_LAST : BOOL;
END_VAR
// press-station: the feeder drops a part into the clamped nest, the press comes down onto it
// and holds for the press time, comes up, the nest unclamps and the ejector pushes the part
// off the nest onto the chute into the bin. Repeat until STOP. The same sequence runs without
// a PLC in press-station.ctl.js.
//
// The clamp goes on BEFORE the feed: a nest that holds the part locates it square on the pocket
// floor, so the press stroke meets it where the drawing says.
//
// Waiting steps wait for an INVARIANT, not for a counter to move: every part fed has reached
// the bin.
//
// The panel has a selector AUTO / INDIVIDUAL: START only in AUTO, the individual buttons only in
// INDIVIDUAL, and a change while the sequence runs is a FAULT, not a pause.

START_EDGE := PB_START AND NOT PB_START_LAST;
PB_START_LAST := PB_START;
IF PB_CSTOP THEN
	STOP_REQ := TRUE;
END_IF;
SEL_CHANGED := SEL_AUTO <> SEL_LAST;
SEL_LAST := SEL_AUTO;

// The master circuit, as on the cell panel: E-STOP is a latching mushroom, MASTER ON energises
// the machine, and nothing runs without it. An E-STOP also loses the home position.
ESTOP := PB_ESTOP;
MASTER_EDGE := PB_MASTER AND NOT PB_MASTER_LAST;
PB_MASTER_LAST := PB_MASTER;
HOME_EDGE := PB_HOME AND NOT PB_HOME_LAST;
PB_HOME_LAST := PB_HOME;
IF ESTOP THEN
	MASTER_ON := FALSE;
	HOMED := FALSE;
ELSIF MASTER_EDGE THEN
	MASTER_ON := TRUE;
END_IF;
READY := MASTER_ON AND NOT ESTOP;

// A write-off goes STALE when the part turns up after all, and then RM + GONE runs PAST EM and
// the step waiting on that invariant stops waiting at all. GONE is a UDINT, so the subtraction
// underflows to about 4 billion when RM is ahead: guard before you subtract.
IF RM_CNT >= EM_CNT THEN
	GONE := 0;
ELSIF RM_CNT + GONE > EM_CNT THEN
	GONE := EM_CNT - RM_CNT;
END_IF;
CASE ST1_STEP OF
	0:	// idle: press up, ejector back, nest free
		CLAMP := FALSE;
		EM_EMIT := FALSE;
		SOL_EJECT := FALSE;
		SOL_P_DN := FALSE;
		SOL_P_UP := TRUE;
		IF START_EDGE AND SEL_AUTO AND READY AND HOMED AND AS_P_UP AND AS_EJ_BACK THEN
			STOP_REQ := FALSE;
			EM_LAST := EM_CNT;
			ST1_STEP := 10;
		END_IF;
	10:	// clamp, then feed one part into the nest
		CLAMP := TRUE;
		EM_EMIT := TRUE;
		IF EM_CNT <> EM_LAST THEN
			EM_EMIT := FALSE;
			ST1_STEP := 20;
		END_IF;
	20:	// the nest reports the part
		IF NEST_P THEN
			ST1_STEP := 30;
		END_IF;
	30:	// press down
		SOL_P_UP := FALSE;
		SOL_P_DN := TRUE;
		IF AS_P_DN THEN
			ST1_STEP := 40;
		END_IF;
	40:	// press time
		IF T_PRESS.Q THEN
			ST1_STEP := 50;
		END_IF;
	50:	// press up
		SOL_P_DN := FALSE;
		SOL_P_UP := TRUE;
		IF AS_P_UP THEN
			ST1_STEP := 60;
		END_IF;
	60:	// unclamp and eject onto the chute
		CLAMP := FALSE;
		SOL_EJECT := TRUE;
		IF AS_EJ_OUT THEN
			ST1_STEP := 70;
		END_IF;
	70:	// ejector back, and every part fed has reached the bin
		SOL_EJECT := FALSE;
		IF AS_EJ_BACK AND (RM_CNT + GONE >= EM_CNT) THEN
			ST1_STEP := 80;
		END_IF;
	80:	// cycle complete
		CYCLE_CNT := CYCLE_CNT + 1;
		IF STOP_REQ THEN
			ST1_STEP := 0;
		ELSE
			EM_LAST := EM_CNT;
			ST1_STEP := 10;
		END_IF;
	800:	// HOME: press up, ejector back. The clamp is left alone: a real machine does not drop the part it holds
		EM_EMIT := FALSE;
		SOL_EJECT := FALSE;
		SOL_P_DN := FALSE;
		SOL_P_UP := TRUE;
		IF AS_P_UP AND AS_EJ_BACK THEN
			HOMED := TRUE;
			ST1_STEP := 0;
		END_IF;
	910:	// E-STOP: the master circuit is open, so every solenoid de-energises - which is what
		// really happens: a 5/2 single-solenoid valve springs back, a double one holds. The holders keep their parts: a real machine does not let go when the power drops.
		EM_EMIT := FALSE;
		SOL_P_DN := FALSE;
		SOL_P_UP := FALSE;
		SOL_EJECT := FALSE;
		IF READY THEN	// MASTER ON after the mushroom is released
			ST1_STEP := 0;
		END_IF;
	900:	// FAULT: a step stopped moving (part taken out of the nest, never arrived, never reached
		// the bin), or the selector was turned while running. Feeding off, press up, ejector
		// back; the clamp keeps whatever it holds.
		EM_EMIT := FALSE;
		SOL_EJECT := FALSE;
		SOL_P_DN := FALSE;
		SOL_P_UP := TRUE;
		IF START_EDGE AND SEL_AUTO THEN
			STOP_REQ := FALSE;
			// Acknowledging writes off whatever never reached the bin. Only HERE.
			GONE := EM_CNT - RM_CNT;
			ST1_STEP := 0;
		END_IF;
END_CASE;

T_PRESS(In := (ST1_STEP = 40), PT := T#500ms);

// Watchdog: a running step that stops moving is a jam, not patience. A selector change while
// running trips the same way.
T_WD(In := (ST1_STEP = STEP_LAST) AND (ST1_STEP <> 0) AND (ST1_STEP <> 900) AND (ST1_STEP <> 910), PT := T#15s);
IF ST1_STEP <> STEP_LAST THEN
	STEP_LAST := ST1_STEP;
END_IF;
IF T_WD.Q OR (SEL_CHANGED AND (ST1_STEP <> 0) AND (ST1_STEP <> 900) AND (ST1_STEP <> 910)) THEN
	ST1_STEP := 900;
	EM_EMIT := FALSE;
	SOL_EJECT := FALSE;
	SOL_P_DN := FALSE;
	SOL_P_UP := TRUE;
END_IF;

// E-STOP at any moment, and the HOME button when the machine is energised and idle.
IF ESTOP THEN
	IF ST1_STEP <> 910 THEN
		ST1_STEP := 910;
	END_IF;
	EM_EMIT := FALSE;
	SOL_P_DN := FALSE;
	SOL_P_UP := FALSE;
	SOL_EJECT := FALSE;
ELSIF HOME_EDGE AND READY AND (ST1_STEP = 0) THEN
	ST1_STEP := 800;
END_IF;

AUTO_RUN := (ST1_STEP <> 0) AND (ST1_STEP <> 800) AND (ST1_STEP <> 900) AND (ST1_STEP <> 910);

// Individual operation: momentary buttons, a PLC toggle memory per actuator, cleared when INDIVIDUAL
// ends. The feed button pulses one part.
IF NOT SEL_AUTO AND NOT AUTO_RUN AND READY AND (ST1_STEP <> 800) THEN
	IF IND_CLAMP AND NOT IND_CLAMP_LAST THEN
		MEM_CLAMP := NOT MEM_CLAMP;
	END_IF;
	IF IND_PRESS AND NOT IND_PRESS_LAST THEN
		MEM_PRESS := NOT MEM_PRESS;
	END_IF;
	IF IND_EJECT AND NOT IND_EJECT_LAST THEN
		MEM_EJECT := NOT MEM_EJECT;
	END_IF;
	EM_EMIT := IND_FEED;
	CLAMP := MEM_CLAMP;
	SOL_P_DN := MEM_PRESS;
	SOL_P_UP := NOT MEM_PRESS;
	SOL_EJECT := MEM_EJECT;
ELSE
	MEM_CLAMP := FALSE;
	MEM_PRESS := FALSE;
	MEM_EJECT := FALSE;
END_IF;
IND_CLAMP_LAST := IND_CLAMP;
IND_PRESS_LAST := IND_PRESS;
IND_EJECT_LAST := IND_EJECT;

PL_START := AUTO_RUN;
PL_MASTER := MASTER_ON;
PL_HOME := HOMED;

(* ---- robot-pitch.st ---- *)
VAR
	START_EDGE : BOOL;
	PB_START_LAST : BOOL;
	STOP_REQ : BOOL;
	SEL_LAST : BOOL := TRUE;
	SEL_CHANGED : BOOL;
	T_WD : TON;
	T_PICK : TON;
	T_DROP : TON;
	T_PROC : TON;
	T_FILL : TON;
	STEP_LAST : UDINT;
	ROW : UINT;
	NEED_FILL : BOOL := TRUE;
	PAL_BASE : UDINT;
	FILL_MOVED : BOOL;
	PICKED : BOOL;
	ALL_DONE : BOOL;
	ALL_CLEAR : BOOL;
	ANY_VAC : BOOL;
	NO_VAC : BOOL;
	PAL_UP_1 : LREAL;
	PAL_UP_2 : LREAL;
	PAL_UP_3 : LREAL;
	PAL_UP_4 : LREAL;
	PAL_UP_5 : LREAL;
	PAL_UP_6 : LREAL;
	PAL_AT_1 : LREAL;
	PAL_AT_2 : LREAL;
	PAL_AT_3 : LREAL;
	PAL_AT_4 : LREAL;
	PAL_AT_5 : LREAL;
	PAL_AT_6 : LREAL;
	MEM_VAC : BOOL;
	IND_VAC_LAST : BOOL;
	IND_ACTIVE : BOOL;
	ESTOP : BOOL;
	READY : BOOL;
	MASTER_ON : BOOL;
	HOMED : BOOL;
	MASTER_EDGE : BOOL;
	PB_MASTER_LAST : BOOL;
	HOME_EDGE : BOOL;
	PB_HOME_LAST : BOOL;
END_VAR
// robot-pitch: a FANUC LR Mate 200iD with a cam-driven pitch-change head. Five cups take a ROW
// of five plugs from the 5 x 5 pallet at 100 mm pitch, the cam closes them to 60 mm, the row is
// set into the five-pocket jig, the jig does its process, and the row is picked again at 60 and
// dropped into the bin. One cycle = one row. The same sequence runs without a PLC in
// robot-pitch.ctl.js.
//
// The poses are joint angles solved once against the scene's kinematics (0.05 mm, >= 30 deg of
// margin to every limit). Moves are joint-space: six targets and Executes together, wait for
// every Done, then drop Execute and wait for Done to clear before the next move.
//
// The panel has a selector AUTO / INDIVIDUAL (rb4axis): START only in AUTO, the individual
// buttons only in INDIVIDUAL, and a change while the sequence runs is a FAULT, not a pause.

START_EDGE := PB_START AND NOT PB_START_LAST;
PB_START_LAST := PB_START;
IF PB_CSTOP THEN
	STOP_REQ := TRUE;
END_IF;
SEL_CHANGED := SEL_AUTO <> SEL_LAST;
SEL_LAST := SEL_AUTO;

// The master circuit, as on the cell panel: E-STOP is a latching mushroom, MASTER ON energises
// the machine, and nothing runs without it. An E-STOP also loses the home position.
ESTOP := PB_ESTOP;
MASTER_EDGE := PB_MASTER AND NOT PB_MASTER_LAST;
PB_MASTER_LAST := PB_MASTER;
HOME_EDGE := PB_HOME AND NOT PB_HOME_LAST;
PB_HOME_LAST := PB_HOME;
IF ESTOP THEN
	MASTER_ON := FALSE;
	HOMED := FALSE;
ELSIF MASTER_EDGE THEN
	MASTER_ON := TRUE;
END_IF;
READY := MASTER_ON AND NOT ESTOP;

ALL_DONE := J1_DONE AND J2_DONE AND J3_DONE AND J4_DONE AND J5_DONE AND J6_DONE;
ALL_CLEAR := NOT J1_DONE AND NOT J2_DONE AND NOT J3_DONE AND NOT J4_DONE AND NOT J5_DONE AND NOT J6_DONE;
ANY_VAC := VAC_C0 OR VAC_C1 OR VAC_C2 OR VAC_C3 OR VAC_C4;
NO_VAC := NOT ANY_VAC;

// The pallet row's poses, from the table (a lookup, not a step of the sequence)
CASE ROW OF
	0:
		PAL_UP_1 := -26.56;
		PAL_UP_2 := 11.48;
		PAL_UP_3 := -4.65;
		PAL_UP_4 := 0.01;
		PAL_UP_5 := -73.87;
		PAL_UP_6 := 26.55;
		PAL_AT_1 := -26.57;
		PAL_AT_2 := 16.99;
		PAL_AT_3 := -15.72;
		PAL_AT_4 := -0.01;
		PAL_AT_5 := -57.29;
		PAL_AT_6 := 26.58;
	1:
		PAL_UP_1 := -14.03;
		PAL_UP_2 := 5.51;
		PAL_UP_3 := -11.49;
		PAL_UP_4 := 0.01;
		PAL_UP_5 := -73.00;
		PAL_UP_6 := 14.02;
		PAL_AT_1 := -14.04;
		PAL_AT_2 := 11.47;
		PAL_AT_3 := -22.74;
		PAL_AT_4 := -0.01;
		PAL_AT_5 := -55.79;
		PAL_AT_6 := 14.05;
	2:
		PAL_UP_1 := 0.00;
		PAL_UP_2 := 3.41;
		PAL_UP_3 := -13.75;
		PAL_UP_4 := 0.00;
		PAL_UP_5 := -72.85;
		PAL_UP_6 := 0.00;
		PAL_AT_1 := 0.00;
		PAL_AT_2 := 9.49;
		PAL_AT_3 := -25.11;
		PAL_AT_4 := 0.00;
		PAL_AT_5 := -55.40;
		PAL_AT_6 := 0.00;
	3:
		PAL_UP_1 := 14.03;
		PAL_UP_2 := 5.51;
		PAL_UP_3 := -11.49;
		PAL_UP_4 := -0.01;
		PAL_UP_5 := -73.00;
		PAL_UP_6 := -14.02;
		PAL_AT_1 := 14.04;
		PAL_AT_2 := 11.47;
		PAL_AT_3 := -22.74;
		PAL_AT_4 := 0.01;
		PAL_AT_5 := -55.79;
		PAL_AT_6 := -14.05;
	4:
		PAL_UP_1 := 26.56;
		PAL_UP_2 := 11.48;
		PAL_UP_3 := -4.65;
		PAL_UP_4 := -0.01;
		PAL_UP_5 := -73.87;
		PAL_UP_6 := -26.55;
		PAL_AT_1 := 26.57;
		PAL_AT_2 := 16.99;
		PAL_AT_3 := -15.72;
		PAL_AT_4 := 0.01;
		PAL_AT_5 := -57.29;
		PAL_AT_6 := -26.58;
END_CASE;

// The pallet is FULL when the loader stops delivering: the timer restarts on every plug.
FILL_MOVED := EM_PAL_CNT <> PAL_BASE;
IF FILL_MOVED THEN
	PAL_BASE := EM_PAL_CNT;
END_IF;

CASE ST1_STEP OF
	0:	// idle
		J1_EXEC := FALSE;
		J2_EXEC := FALSE;
		J3_EXEC := FALSE;
		J4_EXEC := FALSE;
		J5_EXEC := FALSE;
		J6_EXEC := FALSE;
		CAM_EXEC := FALSE;
		EM_PAL_EN := FALSE;
		VAC_ON := FALSE;
		PAL_CLAMP := TRUE;
		JIG_CLAMP := TRUE;
		IF START_EDGE AND SEL_AUTO AND READY AND HOMED THEN
			STOP_REQ := FALSE;
			IF NEED_FILL THEN
				PAL_BASE := EM_PAL_CNT;
				ST1_STEP := 5;
			ELSE
				ST1_STEP := 10;
			END_IF;
		END_IF;
	5:	// a fresh pallet: full when the loader has delivered nothing for 600 ms
		PAL_CLAMP := TRUE;
		EM_PAL_EN := TRUE;
		IF T_FILL.Q THEN
			EM_PAL_EN := FALSE;
			NEED_FILL := FALSE;
			ROW := 0;
			ST1_STEP := 10;
		END_IF;
	10:	// cam wide, above the row
		J1_TGT := PAL_UP_1;
		J2_TGT := PAL_UP_2;
		J3_TGT := PAL_UP_3;
		J4_TGT := PAL_UP_4;
		J5_TGT := PAL_UP_5;
		J6_TGT := PAL_UP_6;
		J1_EXEC := TRUE;
		J2_EXEC := TRUE;
		J3_EXEC := TRUE;
		J4_EXEC := TRUE;
		J5_EXEC := TRUE;
		J6_EXEC := TRUE;
		CAM_TGT := 0.00;
		CAM_EXEC := TRUE;
		IF ALL_DONE AND CAM_DONE THEN
			ST1_STEP := 11;
		END_IF;
	11:
		J1_EXEC := FALSE;
		J2_EXEC := FALSE;
		J3_EXEC := FALSE;
		J4_EXEC := FALSE;
		J5_EXEC := FALSE;
		J6_EXEC := FALSE;
		CAM_EXEC := FALSE;
		IF ALL_CLEAR AND NOT CAM_DONE THEN
			ST1_STEP := 12;
		END_IF;
	12:	// down onto the row
		J1_TGT := PAL_AT_1;
		J2_TGT := PAL_AT_2;
		J3_TGT := PAL_AT_3;
		J4_TGT := PAL_AT_4;
		J5_TGT := PAL_AT_5;
		J6_TGT := PAL_AT_6;
		J1_EXEC := TRUE;
		J2_EXEC := TRUE;
		J3_EXEC := TRUE;
		J4_EXEC := TRUE;
		J5_EXEC := TRUE;
		J6_EXEC := TRUE;
		IF ALL_DONE THEN
			ST1_STEP := 13;
		END_IF;
	13:
		J1_EXEC := FALSE;
		J2_EXEC := FALSE;
		J3_EXEC := FALSE;
		J4_EXEC := FALSE;
		J5_EXEC := FALSE;
		J6_EXEC := FALSE;
		IF ALL_CLEAR THEN
			ST1_STEP := 14;
		END_IF;
	14:	// the pallet lets go, the cups take what is there
		PAL_CLAMP := FALSE;
		VAC_ON := TRUE;
		IF T_PICK.Q THEN
			PICKED := ANY_VAC;
			ST1_STEP := 15;
		END_IF;
	15:	// up with the row
		PAL_CLAMP := TRUE;
		J1_TGT := PAL_UP_1;
		J2_TGT := PAL_UP_2;
		J3_TGT := PAL_UP_3;
		J4_TGT := PAL_UP_4;
		J5_TGT := PAL_UP_5;
		J6_TGT := PAL_UP_6;
		J1_EXEC := TRUE;
		J2_EXEC := TRUE;
		J3_EXEC := TRUE;
		J4_EXEC := TRUE;
		J5_EXEC := TRUE;
		J6_EXEC := TRUE;
		IF ALL_DONE THEN
			ST1_STEP := 16;
		END_IF;
	16:
		J1_EXEC := FALSE;
		J2_EXEC := FALSE;
		J3_EXEC := FALSE;
		J4_EXEC := FALSE;
		J5_EXEC := FALSE;
		J6_EXEC := FALSE;
		IF ALL_CLEAR THEN
			IF PICKED THEN
				ST1_STEP := 17;
			ELSE
				ST1_STEP := 36;
			END_IF;
		END_IF;
	17:	// cam narrow, above the jig
		J1_TGT := 77.47;
		J2_TGT := 13.83;
		J3_TGT := -1.79;
		J4_TGT := 0.00;
		J5_TGT := -74.38;
		J6_TGT := -77.47;
		J1_EXEC := TRUE;
		J2_EXEC := TRUE;
		J3_EXEC := TRUE;
		J4_EXEC := TRUE;
		J5_EXEC := TRUE;
		J6_EXEC := TRUE;
		CAM_TGT := 90.00;
		CAM_EXEC := TRUE;
		IF ALL_DONE AND CAM_DONE THEN
			ST1_STEP := 18;
		END_IF;
	18:
		J1_EXEC := FALSE;
		J2_EXEC := FALSE;
		J3_EXEC := FALSE;
		J4_EXEC := FALSE;
		J5_EXEC := FALSE;
		J6_EXEC := FALSE;
		CAM_EXEC := FALSE;
		IF ALL_CLEAR AND NOT CAM_DONE THEN
			ST1_STEP := 19;
		END_IF;
	19:	// down into the jig
		J1_TGT := 77.47;
		J2_TGT := 19.16;
		J3_TGT := -12.81;
		J4_TGT := 0.00;
		J5_TGT := -58.04;
		J6_TGT := -77.48;
		J1_EXEC := TRUE;
		J2_EXEC := TRUE;
		J3_EXEC := TRUE;
		J4_EXEC := TRUE;
		J5_EXEC := TRUE;
		J6_EXEC := TRUE;
		IF ALL_DONE THEN
			ST1_STEP := 20;
		END_IF;
	20:
		J1_EXEC := FALSE;
		J2_EXEC := FALSE;
		J3_EXEC := FALSE;
		J4_EXEC := FALSE;
		J5_EXEC := FALSE;
		J6_EXEC := FALSE;
		IF ALL_CLEAR THEN
			ST1_STEP := 21;
		END_IF;
	21:	// the jig takes the row
		JIG_CLAMP := TRUE;
		VAC_ON := FALSE;
		IF T_DROP.Q THEN
			ST1_STEP := 22;
		END_IF;
	22:
		J1_TGT := 77.47;
		J2_TGT := 13.83;
		J3_TGT := -1.79;
		J4_TGT := 0.00;
		J5_TGT := -74.38;
		J6_TGT := -77.47;
		J1_EXEC := TRUE;
		J2_EXEC := TRUE;
		J3_EXEC := TRUE;
		J4_EXEC := TRUE;
		J5_EXEC := TRUE;
		J6_EXEC := TRUE;
		IF ALL_DONE THEN
			ST1_STEP := 23;
		END_IF;
	23:
		J1_EXEC := FALSE;
		J2_EXEC := FALSE;
		J3_EXEC := FALSE;
		J4_EXEC := FALSE;
		J5_EXEC := FALSE;
		J6_EXEC := FALSE;
		IF ALL_CLEAR THEN
			ST1_STEP := 24;
		END_IF;
	24:	// the jig does its work
		IF T_PROC.Q THEN
			ST1_STEP := 25;
		END_IF;
	25:	// back down for the finished row
		J1_TGT := 77.47;
		J2_TGT := 19.16;
		J3_TGT := -12.81;
		J4_TGT := 0.00;
		J5_TGT := -58.04;
		J6_TGT := -77.48;
		J1_EXEC := TRUE;
		J2_EXEC := TRUE;
		J3_EXEC := TRUE;
		J4_EXEC := TRUE;
		J5_EXEC := TRUE;
		J6_EXEC := TRUE;
		IF ALL_DONE THEN
			ST1_STEP := 26;
		END_IF;
	26:
		J1_EXEC := FALSE;
		J2_EXEC := FALSE;
		J3_EXEC := FALSE;
		J4_EXEC := FALSE;
		J5_EXEC := FALSE;
		J6_EXEC := FALSE;
		IF ALL_CLEAR THEN
			ST1_STEP := 27;
		END_IF;
	27:	// the jig lets go, the cups take the row
		JIG_CLAMP := FALSE;
		VAC_ON := TRUE;
		IF T_PICK.Q THEN
			PICKED := ANY_VAC;
			ST1_STEP := 28;
		END_IF;
	28:
		JIG_CLAMP := TRUE;
		J1_TGT := 77.47;
		J2_TGT := 13.83;
		J3_TGT := -1.79;
		J4_TGT := 0.00;
		J5_TGT := -74.38;
		J6_TGT := -77.47;
		J1_EXEC := TRUE;
		J2_EXEC := TRUE;
		J3_EXEC := TRUE;
		J4_EXEC := TRUE;
		J5_EXEC := TRUE;
		J6_EXEC := TRUE;
		IF ALL_DONE THEN
			ST1_STEP := 29;
		END_IF;
	29:
		J1_EXEC := FALSE;
		J2_EXEC := FALSE;
		J3_EXEC := FALSE;
		J4_EXEC := FALSE;
		J5_EXEC := FALSE;
		J6_EXEC := FALSE;
		IF ALL_CLEAR THEN
			ST1_STEP := 30;
		END_IF;
	30:	// over the bin
		J1_TGT := 46.97;
		J2_TGT := 46.74;
		J3_TGT := 55.89;
		J4_TGT := 0.00;
		J5_TGT := -99.14;
		J6_TGT := -46.97;
		J1_EXEC := TRUE;
		J2_EXEC := TRUE;
		J3_EXEC := TRUE;
		J4_EXEC := TRUE;
		J5_EXEC := TRUE;
		J6_EXEC := TRUE;
		IF ALL_DONE THEN
			ST1_STEP := 31;
		END_IF;
	31:
		J1_EXEC := FALSE;
		J2_EXEC := FALSE;
		J3_EXEC := FALSE;
		J4_EXEC := FALSE;
		J5_EXEC := FALSE;
		J6_EXEC := FALSE;
		IF ALL_CLEAR THEN
			ST1_STEP := 32;
		END_IF;
	32:	// drop
		VAC_ON := FALSE;
		IF T_DROP.Q THEN
			ST1_STEP := 33;
		END_IF;
	33:	// cam wide again for the next row
		CAM_TGT := 0.00;
		CAM_EXEC := TRUE;
		IF CAM_DONE THEN
			ST1_STEP := 34;
		END_IF;
	34:
		CAM_EXEC := FALSE;
		IF NOT CAM_DONE THEN
			ST1_STEP := 35;
		END_IF;
	35:	// cycle complete: one row
		CYCLE_CNT := CYCLE_CNT + 1;
		ROW := ROW + 1;
		IF ROW >= 5 THEN
			ROW := 0;
			NEED_FILL := TRUE;
		END_IF;
		IF STOP_REQ THEN
			ST1_STEP := 0;
		ELSIF NEED_FILL THEN
			PAL_BASE := EM_PAL_CNT;
			ST1_STEP := 5;
		ELSE
			ST1_STEP := 10;
		END_IF;
	36:	// nothing came up from this row: not a cycle
		ROW := ROW + 1;
		IF ROW >= 5 THEN
			ROW := 0;
			NEED_FILL := TRUE;
		END_IF;
		IF STOP_REQ THEN
			ST1_STEP := 0;
		ELSIF NEED_FILL THEN
			PAL_BASE := EM_PAL_CNT;
			ST1_STEP := 5;
		ELSE
			ST1_STEP := 10;
		END_IF;
	800:	// HOME: the arm to its travel pose, the cam wide; the cups keep what they hold
		EM_PAL_EN := FALSE;
		J1_TGT := 0.00;
		J2_TGT := 0.00;
		J3_TGT := 0.00;
		J4_TGT := 0.00;
		J5_TGT := -90.00;
		J6_TGT := 0.00;
		J1_EXEC := TRUE;
		J2_EXEC := TRUE;
		J3_EXEC := TRUE;
		J4_EXEC := TRUE;
		J5_EXEC := TRUE;
		J6_EXEC := TRUE;
		CAM_TGT := 0.00;
		CAM_EXEC := TRUE;
		IF ALL_DONE AND CAM_DONE THEN
			J1_EXEC := FALSE;
			J2_EXEC := FALSE;
			J3_EXEC := FALSE;
			J4_EXEC := FALSE;
			J5_EXEC := FALSE;
			J6_EXEC := FALSE;
			CAM_EXEC := FALSE;
			EM_PAL_EN := FALSE;
			HOMED := TRUE;
			ST1_STEP := 0;
		END_IF;
	910:	// E-STOP: the master circuit is open, every drive stops where it is. The cups KEEP
		// their plugs: five plugs let go over the pallet is not what a real head does.
		J1_EXEC := FALSE;
		J2_EXEC := FALSE;
		J3_EXEC := FALSE;
		J4_EXEC := FALSE;
		J5_EXEC := FALSE;
		J6_EXEC := FALSE;
		CAM_EXEC := FALSE;
		EM_PAL_EN := FALSE;
		IF READY THEN	// MASTER ON after the mushroom is released
			ST1_STEP := 0;
		END_IF;
	900:	// FAULT: a step stopped moving, or the selector was turned while running.
		J1_EXEC := FALSE;
		J2_EXEC := FALSE;
		J3_EXEC := FALSE;
		J4_EXEC := FALSE;
		J5_EXEC := FALSE;
		J6_EXEC := FALSE;
		CAM_EXEC := FALSE;
		EM_PAL_EN := FALSE;
		IF START_EDGE AND SEL_AUTO THEN
			STOP_REQ := FALSE;
			ST1_STEP := 0;
		END_IF;
END_CASE;

T_PICK(In := (ST1_STEP = 14) OR (ST1_STEP = 27), PT := T#600ms);
T_DROP(In := ((ST1_STEP = 21) OR (ST1_STEP = 32)) AND NO_VAC, PT := T#300ms);
T_PROC(In := (ST1_STEP = 24), PT := T#1s);
T_FILL(In := (ST1_STEP = 5) AND NOT FILL_MOVED, PT := T#600ms);

// Watchdog: a running step that stops moving is a jam, not patience. A selector change while
// running trips the same way.
T_WD(In := (ST1_STEP = STEP_LAST) AND (ST1_STEP <> 0) AND (ST1_STEP <> 900) AND (ST1_STEP <> 910), PT := T#15s);
IF ST1_STEP <> STEP_LAST THEN
	STEP_LAST := ST1_STEP;
END_IF;
IF T_WD.Q OR (SEL_CHANGED AND (ST1_STEP <> 0) AND (ST1_STEP <> 900) AND (ST1_STEP <> 910)) THEN
	ST1_STEP := 900;
	J1_EXEC := FALSE;
	J2_EXEC := FALSE;
	J3_EXEC := FALSE;
	J4_EXEC := FALSE;
	J5_EXEC := FALSE;
	J6_EXEC := FALSE;
	CAM_EXEC := FALSE;
	EM_PAL_EN := FALSE;
END_IF;

// E-STOP at any moment, and the HOME button when the machine is energised and idle.
IF ESTOP THEN
	IF ST1_STEP <> 910 THEN
		ST1_STEP := 910;
	END_IF;
	J1_EXEC := FALSE;
	J2_EXEC := FALSE;
	J3_EXEC := FALSE;
	J4_EXEC := FALSE;
	J5_EXEC := FALSE;
	J6_EXEC := FALSE;
	CAM_EXEC := FALSE;
	EM_PAL_EN := FALSE;
ELSIF HOME_EDGE AND READY AND (ST1_STEP = 0) THEN
	ST1_STEP := 800;
END_IF;

AUTO_RUN := (ST1_STEP <> 0) AND (ST1_STEP <> 800) AND (ST1_STEP <> 900) AND (ST1_STEP <> 910);

// Individual operation: jog buttons drive the joints straight (the axis holds its limits), the
// cam buttons command an end, the vacuum toggles. Nothing stays latched into AUTO.
IND_ACTIVE := NOT SEL_AUTO AND NOT AUTO_RUN AND READY AND (ST1_STEP <> 800);
J1_JOG_P := IND_ACTIVE AND IND_J1_P;
J1_JOG_N := IND_ACTIVE AND IND_J1_N;
J2_JOG_P := IND_ACTIVE AND IND_J2_P;
J2_JOG_N := IND_ACTIVE AND IND_J2_N;
J3_JOG_P := IND_ACTIVE AND IND_J3_P;
J3_JOG_N := IND_ACTIVE AND IND_J3_N;
J4_JOG_P := IND_ACTIVE AND IND_J4_P;
J4_JOG_N := IND_ACTIVE AND IND_J4_N;
J5_JOG_P := IND_ACTIVE AND IND_J5_P;
J5_JOG_N := IND_ACTIVE AND IND_J5_N;
J6_JOG_P := IND_ACTIVE AND IND_J6_P;
J6_JOG_N := IND_ACTIVE AND IND_J6_N;
IF IND_ACTIVE THEN
	IF IND_VAC AND NOT IND_VAC_LAST THEN
		MEM_VAC := NOT MEM_VAC;
	END_IF;
	VAC_ON := MEM_VAC;
	IF IND_CAM_WIDE THEN
		CAM_TGT := 0.00;
		CAM_EXEC := TRUE;
	ELSIF IND_CAM_NARROW THEN
		CAM_TGT := 90.00;
		CAM_EXEC := TRUE;
	ELSE
		CAM_EXEC := FALSE;
	END_IF;
ELSE
	MEM_VAC := FALSE;
END_IF;
IND_VAC_LAST := IND_VAC;

// The speed override the operator dialled in, passed on to the axes.
OVR := OVR_SET;

PL_START := AUTO_RUN;
PL_MASTER := MASTER_ON;
PL_HOME := HOMED;

(* ---- sort-by-height.st ---- *)
VAR
	START_EDGE : BOOL;
	PB_START_LAST : BOOL;
	STOP_REQ : BOOL;
	TALL_TURN : BOOL;
	EM_T_LAST : UDINT;
	EM_S_LAST : UDINT;
	T_SETTLE : TON;
	T_WD : TON;
	STEP_LAST : UDINT;
	GONE_T : UDINT;
	GONE_S : UDINT;
END_VAR
// sort-by-height: feed a tall part and a short part by turns, stop each one at the beams, and
// sort it by which beams are broken. The low beam sees any part; only a tall part reaches the
// high one. Tall parts are pushed off the belt into the reject chute, short ones ride on to the
// outfeed. The same sequence runs without a PLC in sort-by-height.ctl.js.
//
// Waiting steps wait for INVARIANTS - every tall part emitted has reached the bin, every short
// part the outfeed - and the conveying step first waits for the beam to clear, because a part
// still in it belongs to the last cycle.

START_EDGE := PB_START AND NOT PB_START_LAST;
PB_START_LAST := PB_START;
IF PB_STOP THEN
	STOP_REQ := TRUE;
END_IF;

// A write-off goes STALE when the part turns up after all, and then RM + GONE runs PAST EM and
// the step waiting on that invariant stops waiting at all. GONE_T and GONE_S are UDINTs, so the
// subtraction underflows to about 4 billion when RM is ahead: guard before you subtract.
IF RM_T_CNT >= EM_T_CNT THEN
	GONE_T := 0;
ELSIF RM_T_CNT + GONE_T > EM_T_CNT THEN
	GONE_T := EM_T_CNT - RM_T_CNT;
END_IF;
IF RM_S_CNT >= EM_S_CNT THEN
	GONE_S := 0;
ELSIF RM_S_CNT + GONE_S > EM_S_CNT THEN
	GONE_S := EM_S_CNT - RM_S_CNT;
END_IF;

CASE ST1_STEP OF
	0:	// idle
		CV_RUN := FALSE;
		EM_T_EMIT := FALSE;
		EM_S_EMIT := FALSE;
		SOL_PUSH := FALSE;
		IF START_EDGE AND AS_PUSH_RET THEN
			STOP_REQ := FALSE;
			EM_T_LAST := EM_T_CNT;
			EM_S_LAST := EM_S_CNT;
			ST1_STEP := 10;
		END_IF;
	10:	// feed one part, tall and short by turns
		IF TALL_TURN THEN
			EM_T_EMIT := TRUE;
			IF EM_T_CNT <> EM_T_LAST THEN
				EM_T_EMIT := FALSE;
				ST1_STEP := 15;
			END_IF;
		ELSE
			EM_S_EMIT := TRUE;
			IF EM_S_CNT <> EM_S_LAST THEN
				EM_S_EMIT := FALSE;
				ST1_STEP := 15;
			END_IF;
		END_IF;
	15:	// the beam must be clear before this part runs to it
		CV_RUN := TRUE;
		IF NOT PE_LOW THEN
			ST1_STEP := 20;
		END_IF;
	20:	// carry it to the beams
		CV_RUN := TRUE;
		IF PE_LOW THEN
			CV_RUN := FALSE;
			ST1_STEP := 30;
		END_IF;
	30:	// let it settle in front of the pusher
		IF T_SETTLE.Q THEN
			ST1_STEP := 40;
		END_IF;
	40:	// the high beam tells tall from short
		IF PE_HIGH THEN
			ST1_STEP := 50;
		ELSE
			ST1_STEP := 60;
		END_IF;
	50:	// push the tall part off the belt
		SOL_PUSH := TRUE;
		IF AS_PUSH_EXT THEN
			ST1_STEP := 55;
		END_IF;
	55:	// pusher back, and the part has reached the bin
		SOL_PUSH := FALSE;
		IF AS_PUSH_RET AND (RM_T_CNT + GONE_T >= EM_T_CNT) THEN
			ST1_STEP := 70;
		END_IF;
	60:	// carry the short part to the outfeed
		CV_RUN := TRUE;
		IF RM_S_CNT + GONE_S >= EM_S_CNT THEN
			CV_RUN := FALSE;
			ST1_STEP := 70;
		END_IF;
	70:	// cycle complete, and the other kind next time
		CYCLE_CNT := CYCLE_CNT + 1;
		TALL_TURN := NOT TALL_TURN;
		IF STOP_REQ THEN
			ST1_STEP := 0;
		ELSE
			EM_T_LAST := EM_T_CNT;
			EM_S_LAST := EM_S_CNT;
			ST1_STEP := 10;
		END_IF;
	900:	// FAULT: a step stopped moving, so one of the two invariants above can never hold
		// again. Acknowledging writes off what never arrived - only HERE, never at every
		// START, or a straggler's removal ends the next cycle.
		CV_RUN := FALSE;
		EM_T_EMIT := FALSE;
		EM_S_EMIT := FALSE;
		SOL_PUSH := FALSE;
		IF START_EDGE THEN
			STOP_REQ := FALSE;
			GONE_T := EM_T_CNT - RM_T_CNT;
			GONE_S := EM_S_CNT - RM_S_CNT;
			ST1_STEP := 0;
		END_IF;
END_CASE;

T_SETTLE(In := (ST1_STEP = 30), PT := T#300ms);

// Watchdog: a step that stops moving is a jam, not patience. A part taken off the belt leaves
// this sequence waiting for a beam, or for an invariant that can no longer hold.
T_WD(In := (ST1_STEP = STEP_LAST) AND (ST1_STEP <> 0) AND (ST1_STEP <> 900), PT := T#15s);
IF ST1_STEP <> STEP_LAST THEN
	STEP_LAST := ST1_STEP;
END_IF;
IF T_WD.Q THEN
	ST1_STEP := 900;
	CV_RUN := FALSE;
	EM_T_EMIT := FALSE;
	EM_S_EMIT := FALSE;
	SOL_PUSH := FALSE;
END_IF;

AUTO_RUN := (ST1_STEP <> 0) AND (ST1_STEP <> 900);
PL_START := AUTO_RUN;

(* ---- sort-by-material.st ---- *)
VAR
	START_EDGE : BOOL;
	PB_START_LAST : BOOL;
	STOP_REQ : BOOL;
	SEL_LAST : BOOL := TRUE;
	SEL_CHANGED : BOOL;
	METAL_TURN : BOOL := TRUE;
	METAL : BOOL;
	EM_M_LAST : UDINT;
	EM_P_LAST : UDINT;
	T_SETTLE : TON;
	T_WD : TON;
	STEP_LAST : UDINT;
	GONE_M : UDINT;
	GONE_P : UDINT;
	MEM_CV : BOOL;
	IND_CV_LAST : BOOL;
	MEM_PUSH : BOOL;
	IND_PUSH_LAST : BOOL;
	ESTOP : BOOL;
	READY : BOOL;
	MASTER_ON : BOOL;
	HOMED : BOOL;
	MASTER_EDGE : BOOL;
	PB_MASTER_LAST : BOOL;
	HOME_EDGE : BOOL;
	PB_HOME_LAST : BOOL;
END_VAR
// sort-by-material: feed a steel part and a plastic part by turns. Both look the same to the stop
// beam; only the inductive proximity sensor upstream sees the steel one, and its pulse is LATCHED
// while the belt carries the part to the pusher. Steel is pushed off into the bin, plastic rides
// on to the outfeed. The same sequence runs without a PLC in sort-by-material.ctl.js.
//
// Waiting steps wait for INVARIANTS - every steel part fed has reached the bin, every plastic part
// the outfeed - and the conveying step first waits for the beam to clear, because a part still in
// it belongs to the last cycle.
//
// The panel has a selector AUTO / INDIVIDUAL: START only in AUTO, the individual buttons only in
// INDIVIDUAL, and a change while the sequence runs is a FAULT, not a pause.

START_EDGE := PB_START AND NOT PB_START_LAST;
PB_START_LAST := PB_START;
IF PB_CSTOP THEN
	STOP_REQ := TRUE;
END_IF;
SEL_CHANGED := SEL_AUTO <> SEL_LAST;
SEL_LAST := SEL_AUTO;

// The master circuit, as on the cell panel: E-STOP is a latching mushroom, MASTER ON energises
// the machine, and nothing runs without it. An E-STOP also loses the home position.
ESTOP := PB_ESTOP;
MASTER_EDGE := PB_MASTER AND NOT PB_MASTER_LAST;
PB_MASTER_LAST := PB_MASTER;
HOME_EDGE := PB_HOME AND NOT PB_HOME_LAST;
PB_HOME_LAST := PB_HOME;
IF ESTOP THEN
	MASTER_ON := FALSE;
	HOMED := FALSE;
ELSIF MASTER_EDGE THEN
	MASTER_ON := TRUE;
END_IF;
READY := MASTER_ON AND NOT ESTOP;

// A write-off goes STALE when the part turns up after all, and then RM + GONE runs PAST EM and
// the step waiting on that invariant stops waiting at all. GONE is a UDINT, so the subtraction
// underflows to about 4 billion when RM is ahead: guard before you subtract.
IF RM_M_CNT >= EM_M_CNT THEN
	GONE_M := 0;
ELSIF RM_M_CNT + GONE_M > EM_M_CNT THEN
	GONE_M := EM_M_CNT - RM_M_CNT;
END_IF;
IF RM_P_CNT >= EM_P_CNT THEN
	GONE_P := 0;
ELSIF RM_P_CNT + GONE_P > EM_P_CNT THEN
	GONE_P := EM_P_CNT - RM_P_CNT;
END_IF;
CASE ST1_STEP OF
	0:	// idle
		CV_RUN := FALSE;
		EM_M_EMIT := FALSE;
		EM_P_EMIT := FALSE;
		SOL_PUSH := FALSE;
		IF START_EDGE AND SEL_AUTO AND READY AND HOMED AND AS_PUSH_RET THEN
			STOP_REQ := FALSE;
			EM_M_LAST := EM_M_CNT;
			EM_P_LAST := EM_P_CNT;
			ST1_STEP := 10;
		END_IF;
	10:	// feed one part, steel and plastic by turns; the metal latch starts clean
		METAL := FALSE;
		IF METAL_TURN THEN
			EM_M_EMIT := TRUE;
			IF EM_M_CNT <> EM_M_LAST THEN
				EM_M_EMIT := FALSE;
				ST1_STEP := 15;
			END_IF;
		ELSE
			EM_P_EMIT := TRUE;
			IF EM_P_CNT <> EM_P_LAST THEN
				EM_P_EMIT := FALSE;
				ST1_STEP := 15;
			END_IF;
		END_IF;
	15:	// the beam must be clear before this part runs to it
		CV_RUN := TRUE;
		IF NOT PE_STOP THEN
			ST1_STEP := 20;
		END_IF;
	20:	// carry it past the proximity sensor to the stop beam
		CV_RUN := TRUE;
		IF PE_STOP THEN
			CV_RUN := FALSE;
			ST1_STEP := 30;
		END_IF;
	30:	// let it settle in front of the pusher
		IF T_SETTLE.Q THEN
			ST1_STEP := 40;
		END_IF;
	40:	// the latch says what passed the inductive sensor
		IF METAL THEN
			ST1_STEP := 50;
		ELSE
			ST1_STEP := 60;
		END_IF;
	50:	// push the steel part off the belt
		SOL_PUSH := TRUE;
		IF AS_PUSH_EXT THEN
			ST1_STEP := 55;
		END_IF;
	55:	// pusher back, and every steel part fed has reached the bin
		SOL_PUSH := FALSE;
		IF AS_PUSH_RET AND (RM_M_CNT + GONE_M >= EM_M_CNT) THEN
			ST1_STEP := 70;
		END_IF;
	60:	// carry the plastic part to the outfeed
		CV_RUN := TRUE;
		IF RM_P_CNT + GONE_P >= EM_P_CNT THEN
			CV_RUN := FALSE;
			ST1_STEP := 70;
		END_IF;
	70:	// cycle complete, and the other material next time
		CYCLE_CNT := CYCLE_CNT + 1;
		METAL_TURN := NOT METAL_TURN;
		IF STOP_REQ THEN
			ST1_STEP := 0;
		ELSE
			EM_M_LAST := EM_M_CNT;
			EM_P_LAST := EM_P_CNT;
			ST1_STEP := 10;
		END_IF;
	800:	// HOME: pusher back, belt and feeders off
		CV_RUN := FALSE;
		EM_M_EMIT := FALSE;
		EM_P_EMIT := FALSE;
		SOL_PUSH := FALSE;
		IF AS_PUSH_RET THEN
			HOMED := TRUE;
			ST1_STEP := 0;
		END_IF;
	910:	// E-STOP: the master circuit is open, so every solenoid de-energises - which is what
		// really happens: a 5/2 single-solenoid valve springs back, a double one holds.
		CV_RUN := FALSE;
		EM_M_EMIT := FALSE;
		EM_P_EMIT := FALSE;
		SOL_PUSH := FALSE;
		IF READY THEN	// MASTER ON after the mushroom is released
			ST1_STEP := 0;
		END_IF;
	900:	// FAULT: a step stopped moving (a part taken, jammed, lost or sorted the wrong way), or
		// the selector was turned while running.
		CV_RUN := FALSE;
		EM_M_EMIT := FALSE;
		EM_P_EMIT := FALSE;
		SOL_PUSH := FALSE;
		IF START_EDGE AND SEL_AUTO THEN
			STOP_REQ := FALSE;
			// Acknowledging writes off whatever never reached its bin. Only HERE.
			GONE_M := EM_M_CNT - RM_M_CNT;
			GONE_P := EM_P_CNT - RM_P_CNT;
			ST1_STEP := 0;
		END_IF;
END_CASE;

// The metal latch: the part passes the inductive sensor on its way to the stop beam, so the
// sensor is read while the belt carries it, not when it stands at the pusher.
IF ((ST1_STEP = 15) OR (ST1_STEP = 20)) AND PX_METAL THEN
	METAL := TRUE;
END_IF;

T_SETTLE(In := (ST1_STEP = 30), PT := T#300ms);

// Watchdog: a running step that stops moving is a jam, not patience. A selector change while
// running trips the same way.
T_WD(In := (ST1_STEP = STEP_LAST) AND (ST1_STEP <> 0) AND (ST1_STEP <> 900) AND (ST1_STEP <> 910), PT := T#15s);
IF ST1_STEP <> STEP_LAST THEN
	STEP_LAST := ST1_STEP;
END_IF;
IF T_WD.Q OR (SEL_CHANGED AND (ST1_STEP <> 0) AND (ST1_STEP <> 900) AND (ST1_STEP <> 910)) THEN
	ST1_STEP := 900;
	CV_RUN := FALSE;
	EM_M_EMIT := FALSE;
	EM_P_EMIT := FALSE;
	SOL_PUSH := FALSE;
END_IF;

// E-STOP at any moment, and the HOME button when the machine is energised and idle.
IF ESTOP THEN
	IF ST1_STEP <> 910 THEN
		ST1_STEP := 910;
	END_IF;
	CV_RUN := FALSE;
	EM_M_EMIT := FALSE;
	EM_P_EMIT := FALSE;
	SOL_PUSH := FALSE;
ELSIF HOME_EDGE AND READY AND (ST1_STEP = 0) THEN
	ST1_STEP := 800;
END_IF;

AUTO_RUN := (ST1_STEP <> 0) AND (ST1_STEP <> 800) AND (ST1_STEP <> 900) AND (ST1_STEP <> 910);

// Individual operation: momentary buttons, a PLC toggle memory per actuator, cleared when INDIVIDUAL
// ends. The feed buttons pulse one part each.
IF NOT SEL_AUTO AND NOT AUTO_RUN AND READY AND (ST1_STEP <> 800) THEN
	IF IND_CV AND NOT IND_CV_LAST THEN
		MEM_CV := NOT MEM_CV;
	END_IF;
	IF IND_PUSH AND NOT IND_PUSH_LAST THEN
		MEM_PUSH := NOT MEM_PUSH;
	END_IF;
	CV_RUN := MEM_CV;
	EM_M_EMIT := IND_FEED_M;
	EM_P_EMIT := IND_FEED_P;
	SOL_PUSH := MEM_PUSH;
ELSE
	MEM_CV := FALSE;
	MEM_PUSH := FALSE;
END_IF;
IND_CV_LAST := IND_CV;
IND_PUSH_LAST := IND_PUSH;

// The speed override the operator dialled in, passed on to the axes and the belts.
OVR := OVR_SET;

PL_START := AUTO_RUN;
PL_MASTER := MASTER_ON;
PL_HOME := HOMED;

(* ---- stopper-pusher.st ---- *)
VAR
	START_EDGE : BOOL;
	PB_START_LAST : BOOL;
	STOP_REQ : BOOL;
	SEL_LAST : BOOL := TRUE;
	SEL_CHANGED : BOOL;
	N : UDINT;
	T_SETTLE : TON;
	T_GAP : TON;
	T_WD : TON;
	STEP_LAST : UDINT;
	MEM_CV : BOOL;
	IND_CV_LAST : BOOL;
	MEM_FEED : BOOL;
	IND_FEED_LAST : BOOL;
	MEM_STOP : BOOL;
	IND_STOP_LAST : BOOL;
	MEM_PUSH : BOOL;
	IND_PUSH_LAST : BOOL;
	ESTOP : BOOL;
	READY : BOOL;
	MASTER_ON : BOOL;
	HOMED : BOOL;
	MASTER_EDGE : BOOL;
	PB_MASTER_LAST : BOOL;
	HOME_EDGE : BOOL;
	PB_HOME_LAST : BOOL;
END_VAR
// stopper-pusher: the belt runs, the loader feeds a part every 2.5 s, and a stopper pin holds
// each part at the pusher. Odd parts are pushed off the belt into the reject chute; even parts
// are released to the outfeed. Repeat until STOP. The same sequence runs without a PLC in
// stopper-pusher.ctl.js.
//
// The panel has a selector AUTO / INDIVIDUAL: START only in AUTO, the individual buttons only in
// INDIVIDUAL, and a change while the sequence runs is a FAULT, not a pause.

START_EDGE := PB_START AND NOT PB_START_LAST;
PB_START_LAST := PB_START;
IF PB_CSTOP THEN
	STOP_REQ := TRUE;
END_IF;
SEL_CHANGED := SEL_AUTO <> SEL_LAST;
SEL_LAST := SEL_AUTO;

// The master circuit, as on the cell panel: E-STOP is a latching mushroom, MASTER ON energises
// the machine, and nothing runs without it. An E-STOP also loses the home position.
ESTOP := PB_ESTOP;
MASTER_EDGE := PB_MASTER AND NOT PB_MASTER_LAST;
PB_MASTER_LAST := PB_MASTER;
HOME_EDGE := PB_HOME AND NOT PB_HOME_LAST;
PB_HOME_LAST := PB_HOME;
IF ESTOP THEN
	MASTER_ON := FALSE;
	HOMED := FALSE;
ELSIF MASTER_EDGE THEN
	MASTER_ON := TRUE;
END_IF;
READY := MASTER_ON AND NOT ESTOP;

CASE ST1_STEP OF
	0:	// idle
		CV1_RUN := FALSE;
		EM1_EN := FALSE;
		SOL_STOP := FALSE;
		SOL_PUSH := FALSE;
		IF START_EDGE AND SEL_AUTO AND READY AND HOMED AND AS_PUSH_RET THEN
			STOP_REQ := FALSE;
			ST1_STEP := 10;
		END_IF;
	10:	// stopper down, belt and loader on
		SOL_STOP := TRUE;
		CV1_RUN := TRUE;
		EM1_EN := TRUE;
		IF AS_STOP_DN THEN
			ST1_STEP := 20;
		END_IF;
	20:	// a part settles against the pin
		IF T_SETTLE.Q THEN
			ST1_STEP := 30;
		END_IF;
	30:	// odd parts to the reject chute, even parts to the outfeed
		N := N + 1;
		IF (N MOD 2) = 1 THEN
			ST1_STEP := 40;
		ELSE
			ST1_STEP := 60;
		END_IF;
	40:	// push
		SOL_PUSH := TRUE;
		IF AS_PUSH_EXT THEN
			ST1_STEP := 50;
		END_IF;
	50:	// pusher back, and the part is gone from the eye
		SOL_PUSH := FALSE;
		IF AS_PUSH_RET AND NOT PE_STOP THEN
			ST1_STEP := 80;
		END_IF;
	60:	// release: stopper up until the part has left the eye
		SOL_STOP := FALSE;
		IF NOT PE_STOP THEN
			ST1_STEP := 70;
		END_IF;
	70:	// let it clear the pin, then block again
		IF T_GAP.Q THEN
			SOL_STOP := TRUE;
			IF AS_STOP_DN THEN
				ST1_STEP := 80;
			END_IF;
		END_IF;
	80:	// cycle complete
		CYCLE_CNT := CYCLE_CNT + 1;
		IF STOP_REQ THEN
			ST1_STEP := 0;
		ELSE
			ST1_STEP := 20;
		END_IF;
	800:	// HOME: pusher back, stopper up, belt and loader off
		CV1_RUN := FALSE;
		EM1_EN := FALSE;
		SOL_STOP := FALSE;
		SOL_PUSH := FALSE;
		IF AS_PUSH_RET AND AS_STOP_UP THEN
			HOMED := TRUE;
			ST1_STEP := 0;
		END_IF;
	910:	// E-STOP: the master circuit is open, so every solenoid de-energises - which is what
		// really happens: a 5/2 single-solenoid valve springs back, a double one holds.
		CV1_RUN := FALSE;
		EM1_EN := FALSE;
		SOL_STOP := FALSE;
		SOL_PUSH := FALSE;
		IF READY THEN	// MASTER ON after the mushroom is released
			ST1_STEP := 0;
		END_IF;
	900:	// FAULT: a step stopped moving, or the selector was turned while running.
		CV1_RUN := FALSE;
		EM1_EN := FALSE;
		// LEAVE THE STOPPER DOWN - it is holding the queue back, and a fault that releases it
		// runs the whole queue into a machine that has just stopped. E-STOP is the other case.
		SOL_PUSH := FALSE;
		IF START_EDGE AND SEL_AUTO THEN
			STOP_REQ := FALSE;
			ST1_STEP := 0;
		END_IF;
END_CASE;

T_SETTLE(In := (ST1_STEP = 20) AND PE_STOP, PT := T#300ms);
T_GAP(In := (ST1_STEP = 70), PT := T#400ms);

// Watchdog: a running step that stops moving is a jam, not patience. A selector change while
// running trips the same way.
T_WD(In := (ST1_STEP = STEP_LAST) AND (ST1_STEP <> 0) AND (ST1_STEP <> 900) AND (ST1_STEP <> 910), PT := T#15s);
IF ST1_STEP <> STEP_LAST THEN
	STEP_LAST := ST1_STEP;
END_IF;
IF T_WD.Q OR (SEL_CHANGED AND (ST1_STEP <> 0) AND (ST1_STEP <> 900) AND (ST1_STEP <> 910)) THEN
	ST1_STEP := 900;
	CV1_RUN := FALSE;
	EM1_EN := FALSE;
	// the stopper stays DOWN: it is holding the queue back
	SOL_PUSH := FALSE;
END_IF;

// E-STOP at any moment, and the HOME button when the machine is energised and idle.
IF ESTOP THEN
	IF ST1_STEP <> 910 THEN
		ST1_STEP := 910;
	END_IF;
	CV1_RUN := FALSE;
	EM1_EN := FALSE;
	SOL_STOP := FALSE;
	SOL_PUSH := FALSE;
ELSIF HOME_EDGE AND READY AND (ST1_STEP = 0) THEN
	ST1_STEP := 800;
END_IF;

AUTO_RUN := (ST1_STEP <> 0) AND (ST1_STEP <> 800) AND (ST1_STEP <> 900) AND (ST1_STEP <> 910);

// Individual operation: momentary buttons, a PLC toggle memory per actuator, cleared when INDIVIDUAL ends.
IF NOT SEL_AUTO AND NOT AUTO_RUN AND READY AND (ST1_STEP <> 800) THEN
	IF IND_CV AND NOT IND_CV_LAST THEN
		MEM_CV := NOT MEM_CV;
	END_IF;
	IF IND_FEED AND NOT IND_FEED_LAST THEN
		MEM_FEED := NOT MEM_FEED;
	END_IF;
	IF IND_STOP AND NOT IND_STOP_LAST THEN
		MEM_STOP := NOT MEM_STOP;
	END_IF;
	IF IND_PUSH AND NOT IND_PUSH_LAST THEN
		MEM_PUSH := NOT MEM_PUSH;
	END_IF;
	CV1_RUN := MEM_CV;
	EM1_EN := MEM_FEED;
	SOL_STOP := MEM_STOP;
	SOL_PUSH := MEM_PUSH;
ELSE
	MEM_CV := FALSE;
	MEM_FEED := FALSE;
	MEM_STOP := FALSE;
	MEM_PUSH := FALSE;
END_IF;
IND_CV_LAST := IND_CV;
IND_FEED_LAST := IND_FEED;
IND_STOP_LAST := IND_STOP;
IND_PUSH_LAST := IND_PUSH;

// The speed override the operator dialled in, passed on to the axes and the belts.
OVR := OVR_SET;

PL_START := AUTO_RUN;
PL_MASTER := MASTER_ON;
PL_HOME := HOMED;
